KUKA KRL program: MyProgram_128().src

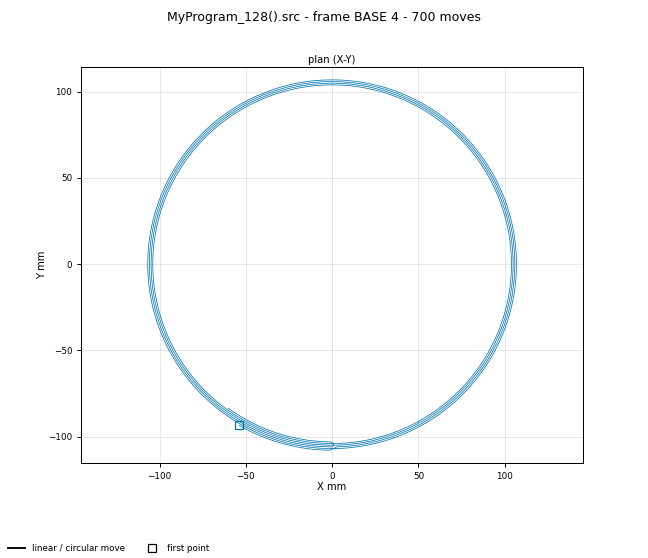
[picture p0: tool path of MyProgram_128().src in frame BASE 4, 700 of 700 moves have a stored position in this frame; points joined in program order, loops and branches not executed]
&ACCESS RVP
&REL 1
&PARAM TEMPLATE = C:\KRC\Roboter\Template\vorgabe
&PARAM EDITMASK = *
DEF MyProgram_128()
; ---- Setting reference (Base) ----
$BASE = BASE_DATA[4]

; --------------------------
; ---- Setting tool (TCP) ----
$TOOL = TOOL_DATA[3]
; --------------------------

$VEL.CP = VEL_APROX_PRINT
Startdeposition()
$VEL.CP = VEL_PRINT
LIN {X -53.8766,Y -93.3824,Z 106,A -123.5845,B 24.9478,C -1.6698,E1 24.9211,E2 209.3121} C_DIS
LIN {X -51.7834,Y -94.56,Z 106,A -122.4157,B 24.9481,C -1.6638,E1 24.9239,E2 208.1542} C_DIS
LIN {X -49.6515,Y -95.6979,Z 106,A -121.0163,B 24.9479,C -1.6666,E1 24.9274,E2 206.7442} C_DIS
LIN {X -46.8609,Y -97.0928,Z 106,A -119.3542,B 24.9481,C -1.6648,E1 24.9316,E2 205.082} C_DIS
LIN {X -43.6897,Y -98.5625,Z 106,A -117.4919,B 24.9481,C -1.6628,E1 24.9363,E2 203.2197} C_DIS
LIN {X -41.2577,Y -99.605,Z 106,A -116.0826,B 24.9483,C -1.6615,E1 24.9399,E2 201.8104} C_DIS
LIN {X -38.8009,Y -100.5875,Z 106,A -114.6732,B 24.9483,C -1.6603,E1 24.9436,E2 200.4009} C_DIS
LIN {X -35.8736,Y -101.6663,Z 106,A -113.2424,B 24.949,C -1.6498,E1 24.9473,E2 198.9921} C_DIS
LIN {X -33.5947,Y -102.4426,Z 106,A -111.8444,B 24.9488,C -1.6534,E1 24.951,E2 197.5829} C_DIS
LIN {X -30.8419,Y -103.3041,Z 106,A -110.1194,B 24.9484,C -1.66,E1 24.9557,E2 195.8392} C_DIS
LIN {X -27.4775,Y -104.2514,Z 106,A -108.3349,B 24.9486,C -1.6559,E1 24.9605,E2 194.0618} C_DIS
LIN {X -24.4492,Y -105.0009,Z 106,A -106.9046,B 24.9492,C -1.6459,E1 24.9643,E2 192.6533} C_DIS
LIN {X -22.329,Y -105.474,Z 106,A -105.5194,B 24.9487,C -1.6546,E1 24.9681,E2 191.2456} C_DIS
LIN {X -19.6263,Y -106.0096,Z 106,A -103.9265,B 24.9484,C -1.6593,E1 24.9725,E2 189.64} C_DIS
LIN {X -15.8193,Y -106.6448,Z 106,A -101.832,B 24.9484,C -1.6604,E1 24.9783,E2 187.5408} C_DIS
LIN {X -12.7268,Y -107.056,Z 106,A -100.4364,B 24.949,C -1.6495,E1 24.9821,E2 186.1701} C_DIS
LIN {X -10.0957,Y -107.3361,Z 106,A -98.9361,B 24.9488,C -1.6532,E1 24.9863,E2 184.6602} C_DIS
LIN {X -7.3812,Y -107.5567,Z 106,A -97.4197,B 24.9486,C -1.656,E1 24.9906,E2 183.1365} C_DIS
LIN {X -3.9682,Y -107.7386,Z 106,A -95.5034,B 24.9483,C -1.6602,E1 24.9959,E2 181.2098} C_DIS
LIN {X -1.323,Y -107.8036,Z 106,A -94.0977,B 24.9483,C -1.6605,E1 24.9999,E2 179.8035} C_DIS
LIN {X -1.323,Y -107.8036,Z 106,A -94.0977,B 24.9483,C -1.6605,E1 24.9999,E2 179.8035} C_DIS
Enddeposition()
LIN {X 0.7537,Y -106.8293,Z 106,A -94.1088,B 24.9501,C -1.6325,E1 24.9997,E2 179.8808} C_DIS
Startdeposition()
$VEL.CP = VEL_PRINT
LIN {X -4.5597,Y -106.7397,Z 106,A -96.7886,B 24.9497,C -1.6389,E1 24.9922,E2 182.546} C_DIS
LIN {X -8.4258,Y -106.5043,Z 106,A -99.1178,B 24.9503,C -1.6288,E1 24.9856,E2 184.8999} C_DIS
LIN {X -12.2598,Y -106.1314,Z 106,A -100.9493,B 24.9497,C -1.6383,E1 24.9806,E2 186.7099} C_DIS
LIN {X -16.8585,Y -105.4999,Z 106,A -103.5719,B 24.95,C -1.6337,E1 24.9733,E2 189.3458} C_DIS
LIN {X -22.5826,Y -104.4233,Z 106,A -106.933,B 24.9505,C -1.6257,E1 24.9641,E2 192.7297} C_DIS
LIN {X -25.8619,Y -103.6611,Z 106,A -108.2155,B 24.9492,C -1.6471,E1 24.9607,E2 193.963} C_DIS
LIN {X -30.0016,Y -102.5389,Z 106,A -110.7389,B 24.9496,C -1.6399,E1 24.9539,E2 196.5076} C_DIS
LIN {X -33.8683,Y -101.3271,Z 106,A -112.9026,B 24.9495,C -1.6419,E1 24.9481,E2 198.6703} C_DIS
LIN {X -37.7546,Y -99.9437,Z 106,A -115.0418,B 24.9492,C -1.6467,E1 24.9425,E2 200.8024} C_DIS
LIN {X -40.9294,Y -98.6879,Z 106,A -117.0692,B 24.9495,C -1.641,E1 24.9373,E2 202.8481} C_DIS
LIN {X -44.6783,Y -97.0474,Z 106,A -120.2088,B 24.9516,C -1.6074,E1 24.9291,E2 206.0752} C_DIS
LIN {X -50.3226,Y -94.2452,Z 106,A -122.6141,B 24.9491,C -1.6488,E1 24.9234,E2 208.3889} C_DIS
LIN {X -53.8043,Y -92.3021,Z 106,A -124.7623,B 24.9489,C -1.6514,E1 24.9181,E2 210.5371} C_DIS
LIN {X -58.2187,Y -89.583,Z 106,A -128.8926,B 24.9517,C -1.6051,E1 24.9082,E2 214.7909} C_DIS
LIN {X -64.5258,Y -85.1515,Z 106,A -131.6457,B 24.9481,C -1.6638,E1 24.9023,E2 217.414} C_DIS
LIN {X -67.7619,Y -82.6008,Z 106,A -133.8259,B 24.9478,C -1.669,E1 24.8975,E2 219.59} C_DIS
LIN {X -70.8575,Y -79.9604,Z 106,A -135.8732,B 24.9472,C -1.6784,E1 24.8932,E2 221.6232} C_DIS
LIN {X -76.0657,Y -75.0211,Z 106,A -139.5928,B 24.9464,C -1.6912,E1 24.8858,E2 225.3276} C_DIS
LIN {X -77.8033,Y -73.2176,Z 106,A -141.1346,B 24.9467,C -1.6867,E1 24.8828,E2 226.8868} C_DIS
LIN {X -80.0433,Y -70.7645,Z 106,A -143.1927,B 24.9471,C -1.6803,E1 24.8789,E2 228.9691} C_DIS
LIN {X -83.2382,Y -66.9754,Z 106,A -146.096,B 24.9473,C -1.6776,E1 24.8737,E2 231.8925} C_DIS
LIN {X -85.3774,Y -64.2251,Z 106,A -147.9105,B 24.9468,C -1.6841,E1 24.8707,E2 233.7001} C_DIS
LIN {X -87.3667,Y -61.4948,Z 106,A -149.2362,B 24.9454,C -1.7066,E1 24.8686,E2 234.9787} C_DIS
LIN {X -89.6712,Y -58.0812,Z 106,A -151.5516,B 24.9454,C -1.7083,E1 24.865,E2 237.3017} C_DIS
LIN {X -91.6677,Y -54.8776,Z 106,A -153.598,B 24.945,C -1.7128,E1 24.862,E2 239.3477} C_DIS
LIN {X -94.7989,Y -49.2714,Z 106,A -156.9611,B 24.9442,C -1.7252,E1 24.8575,E2 242.6992} C_DIS
LIN {X -96.091,Y -46.7001,Z 106,A -158.6935,B 24.9444,C -1.7226,E1 24.8553,E2 244.4471} C_DIS
LIN {X -97.5751,Y -43.5135,Z 106,A -160.5489,B 24.944,C -1.729,E1 24.8532,E2 246.2973} C_DIS
LIN {X -98.9301,Y -40.336,Z 106,A -162.3903,B 24.9436,C -1.7348,E1 24.8512,E2 248.1351} C_DIS
LIN {X -100.5391,Y -36.142,Z 106,A -165.3865,B 24.9445,C -1.7206,E1 24.8483,E2 251.1821} C_DIS
LIN {X -101.8368,Y -32.3055,Z 106,A -167.2873,B 24.9435,C -1.7369,E1 24.8467,E2 253.0548} C_DIS
LIN {X -103.1179,Y -27.944,Z 106,A -169.4189,B 24.9422,C -1.7555,E1 24.8451,E2 255.1546} C_DIS
LIN {X -104.0092,Y -24.4209,Z 106,A -171.4733,B 24.9421,C -1.7577,E1 24.8437,E2 257.2158} C_DIS
LIN {X -104.724,Y -21.1464,Z 106,A -173.1742,B 24.9415,C -1.7668,E1 24.8428,E2 258.905} C_DIS
LIN {X -105.3666,Y -17.6648,Z 106,A -175.1279,B 24.9412,C -1.7708,E1 24.8418,E2 260.8607} C_DIS
LIN {X -105.8765,Y -14.3058,Z 106,A -177.0343,B 24.9411,C -1.7734,E1 24.841,E2 262.7722} C_DIS
LIN {X -106.2835,Y -10.8648,Z 106,A -178.9414,B 24.9408,C -1.7776,E1 24.8405,E2 264.6807} C_DIS
LIN {X -106.6254,Y -6.7385,Z 106,A 178.8379,B 24.9403,C -1.7847,E1 24.84,E2 266.8979} C_DIS
LIN {X -106.7958,Y -2.9825,Z 106,A 176.9449,B 24.9396,C -1.7957,E1 24.8398,E2 268.7761} C_DIS
LIN {X -106.8353,Y 0.6396,Z 106,A 174.8831,B 24.9394,C -1.7977,E1 24.8398,E2 270.8456} C_DIS
LIN {X -106.6524,Y 6.292,Z 106,A 171.4111,B 24.9398,C -1.7917,E1 24.8402,E2 274.3527} C_DIS
LIN {X -106.3816,Y 9.8551,Z 106,A 169.9779,B 24.9382,C -1.8153,E1 24.8406,E2 275.7384} C_DIS
LIN {X -105.9749,Y 13.5463,Z 106,A 167.9438,B 24.9379,C -1.8202,E1 24.8412,E2 277.7729} C_DIS
LIN {X -105.4663,Y 17.0686,Z 106,A 166.0467,B 24.9375,C -1.8267,E1 24.842,E2 279.6657} C_DIS
LIN {X -104.944,Y 20.0236,Z 106,A 164.3886,B 24.9372,C -1.8301,E1 24.8429,E2 281.3254} C_DIS
LIN {X -104.2041,Y 23.5773,Z 106,A 162.302,B 24.9372,C -1.8313,E1 24.8441,E2 283.4215} C_DIS
LIN {X -103.0755,Y 28.1008,Z 106,A 159.897,B 24.9364,C -1.8427,E1 24.8458,E2 285.8133} C_DIS
LIN {X -102.0096,Y 31.7525,Z 106,A 157.8654,B 24.9359,C -1.8494,E1 24.8474,E2 287.8406} C_DIS
LIN {X -100.516,Y 36.206,Z 106,A 155.5457,B 24.9348,C -1.8645,E1 24.8495,E2 290.1376} C_DIS
LIN {X -98.512,Y 41.3469,Z 106,A 152.3947,B 24.9347,C -1.8666,E1 24.8528,E2 293.3012} C_DIS
LIN {X -96.9626,Y 44.8605,Z 106,A 150.3288,B 24.9343,C -1.8726,E1 24.8551,E2 295.3641} C_DIS
LIN {X -95.5,Y 47.8973,Z 106,A 148.3707,B 24.9343,C -1.8726,E1 24.8575,E2 297.3328} C_DIS
LIN {X -93.8185,Y 51.1105,Z 106,A 146.4825,B 24.9337,C -1.8804,E1 24.86,E2 299.2125} C_DIS
LIN {X -91.9159,Y 54.4576,Z 106,A 144.476,B 24.9331,C -1.8885,E1 24.8628,E2 301.2101} C_DIS
LIN {X -90.0123,Y 57.5499,Z 106,A 142.2059,B 24.9336,C -1.8823,E1 24.8662,E2 303.5066} C_DIS
LIN {X -87.3965,Y 61.452,Z 106,A 139.8627,B 24.9326,C -1.8956,E1 24.8699,E2 305.8295} C_DIS
LIN {X -85.1324,Y 64.5512,Z 106,A 137.8079,B 24.9322,C -1.9014,E1 24.8733,E2 307.8805} C_DIS
LIN {X -82.8401,Y 67.4666,Z 106,A 135.7681,B 24.932,C -1.9048,E1 24.8769,E2 309.9218} C_DIS
LIN {X -80.3579,Y 70.4044,Z 106,A 133.8363,B 24.9313,C -1.9149,E1 24.8804,E2 311.8382} C_DIS
LIN {X -78.0201,Y 72.987,Z 106,A 131.9111,B 24.9311,C -1.9175,E1 24.884,E2 313.7657} C_DIS
LIN {X -75.723,Y 75.3681,Z 106,A 130.2361,B 24.9305,C -1.9255,E1 24.8873,E2 315.4289} C_DIS
LIN {X -73.4692,Y 77.5666,Z 106,A 127.978,B 24.9317,C -1.9086,E1 24.8919,E2 317.7366} C_DIS
LIN {X -70.8207,Y 79.9933,Z 106,A 126.0109,B 24.9315,C -1.9115,E1 24.896,E2 319.7045} C_DIS
LIN {X -68.1002,Y 82.32,Z 106,A 124.5718,B 24.9299,C -1.9335,E1 24.899,E2 321.0968} C_DIS
LIN {X -65.2452,Y 84.6004,Z 106,A 122.6715,B 24.9294,C -1.9399,E1 24.9032,E2 322.9889} C_DIS
LIN {X -62.4948,Y 86.6536,Z 106,A 120.7082,B 24.9295,C -1.9391,E1 24.9076,E2 324.9609} C_DIS
LIN {X -59.6356,Y 88.6445,Z 106,A 118.8631,B 24.9292,C -1.9437,E1 24.9118,E2 326.8013} C_DIS
LIN {X -56.8119,Y 90.48,Z 106,A 116.8638,B 24.9294,C -1.94,E1 24.9166,E2 328.8159} C_DIS
LIN {X -53.1715,Y 92.6658,Z 106,A 114.7,B 24.9288,C -1.9483,E1 24.9218,E2 330.9664} C_DIS
LIN {X -49.8424,Y 94.4981,Z 106,A 112.6693,B 24.9286,C -1.952,E1 24.9267,E2 332.9939} C_DIS
LIN {X -46.6974,Y 96.0923,Z 106,A 110.7823,B 24.9283,C -1.9552,E1 24.9315,E2 334.8783} C_DIS
LIN {X -43.2414,Y 97.6968,Z 106,A 108.4552,B 24.9289,C -1.9476,E1 24.9375,E2 337.2292} C_DIS
LIN {X -33.9206,Y 101.3094,Z 106,A 103.3392,B 24.9277,C -1.964,E1 24.9508,E2 342.3169} C_DIS
LIN {X -29.4331,Y 102.7032,Z 106,A 101.1189,B 24.9266,C -1.9783,E1 24.9566,E2 344.507} C_DIS
LIN {X -26.7938,Y 103.4229,Z 106,A 99.4155,B 24.9272,C -1.9707,E1 24.9613,E2 346.2309} C_DIS
LIN {X -23.5828,Y 104.2028,Z 106,A 97.6173,B 24.9272,C -1.9713,E1 24.9661,E2 348.03} C_DIS
LIN {X -19.9636,Y 104.9556,Z 106,A 95.5584,B 24.9272,C -1.9701,E1 24.9718,E2 350.0943} C_DIS
LIN {X -16.1538,Y 105.6089,Z 106,A 93.6037,B 24.9268,C -1.9761,E1 24.9771,E2 352.0365} C_DIS
LIN {X -12.5623,Y 106.096,Z 106,A 91.3704,B 24.9275,C -1.9661,E1 24.9834,E2 354.2952} C_DIS
LIN {X -8.9146,Y 106.4652,Z 106,A 89.0106,B 24.9286,C -1.9518,E1 24.9901,E2 356.6899} C_DIS
LIN {X -4.6596,Y 106.7354,Z 106,A 87.3422,B 24.9268,C -1.9765,E1 24.9946,E2 358.3001} C_DIS
LIN {X 1.7314,Y 106.8233,Z 106,A 84.2326,B 24.9258,C -1.9897,E1 25.0032,E2 361.3784} C_DIS
LIN {X 7.0338,Y 106.6054,Z 106,A 81.2333,B 24.9262,C -1.9838,E1 25.0116,E2 364.3908} C_DIS
LIN {X 12.9512,Y 106.0505,Z 106,A 77.8395,B 24.9268,C -1.9752,E1 25.021,E2 367.8028} C_DIS
LIN {X 16.5164,Y 105.5529,Z 106,A 76.0583,B 24.9264,C -1.9806,E1 25.0259,E2 369.5696} C_DIS
LIN {X 19.8073,Y 104.9856,Z 106,A 74.0743,B 24.9271,C -1.9723,E1 25.0314,E2 371.5712} C_DIS
LIN {X 23.4551,Y 104.2324,Z 106,A 72.1119,B 24.9271,C -1.9727,E1 25.0368,E2 373.5301} C_DIS
LIN {X 26.9434,Y 103.3844,Z 106,A 70.3953,B 24.9265,C -1.9799,E1 25.0414,E2 375.2271} C_DIS
LIN {X 29.9078,Y 102.5667,Z 106,A 68.5867,B 24.9271,C -1.9723,E1 25.0463,E2 377.0505} C_DIS
LIN {X 32.835,Y 101.6662,Z 106,A 66.99,B 24.9271,C -1.9729,E1 25.0505,E2 378.6429} C_DIS
LIN {X 36.1477,Y 100.5373,Z 106,A 65.0474,B 24.9273,C -1.9686,E1 25.0556,E2 380.5918} C_DIS
LIN {X 40.186,Y 98.9912,Z 106,A 62.8015,B 24.9273,C -1.9693,E1 25.0615,E2 382.8313} C_DIS
LIN {X 43.4213,Y 97.6167,Z 106,A 60.1224,B 24.9298,C -1.9351,E1 25.0685,E2 385.5845} C_DIS
LIN {X 47.8384,Y 95.5292,Z 106,A 58.3036,B 24.9277,C -1.9642,E1 25.0729,E2 387.3296} C_DIS
LIN {X 51.0886,Y 93.8304,Z 106,A 56.4015,B 24.9277,C -1.9642,E1 25.0775,E2 389.2263} C_DIS
LIN {X 54.3432,Y 91.9835,Z 106,A 54.3526,B 24.928,C -1.9596,E1 25.0825,E2 391.28} C_DIS
LIN {X 57.4769,Y 90.0591,Z 106,A 52.336,B 24.9284,C -1.9548,E1 25.0873,E2 393.3016} C_DIS
LIN {X 62.2481,Y 86.8297,Z 106,A 49.389,B 24.9284,C -1.9555,E1 25.0941,E2 396.2369} C_DIS
LIN {X 64.5989,Y 85.0966,Z 106,A 47.6628,B 24.929,C -1.9461,E1 25.0979,E2 397.9792} C_DIS
LIN {X 67.8696,Y 82.5116,Z 106,A 45.6524,B 24.9286,C -1.9512,E1 25.1023,E2 399.9698} C_DIS
LIN {X 70.9515,Y 79.8763,Z 106,A 42.9049,B 24.9307,C -1.9232,E1 25.1082,E2 402.7726} C_DIS
LIN {X 73.4992,Y 77.5384,Z 106,A 41.3863,B 24.9299,C -1.9333,E1 25.1112,E2 404.2612} C_DIS
LIN {X 76.148,Y 74.9379,Z 106,A 39.5513,B 24.9298,C -1.9355,E1 25.1148,E2 406.0832} C_DIS
LIN {X 78.2863,Y 72.7037,Z 106,A 37.6743,B 24.9307,C -1.9227,E1 25.1184,E2 407.9824} C_DIS
LIN {X 80.3504,Y 70.4131,Z 106,A 36.1982,B 24.9304,C -1.9264,E1 25.1211,E2 409.4431} C_DIS
LIN {X 82.8244,Y 67.486,Z 106,A 34.1598,B 24.9307,C -1.9222,E1 25.1248,E2 411.4819} C_DIS
LIN {X 85.7964,Y 63.6674,Z 106,A 31.4837,B 24.9314,C -1.9124,E1 25.1293,E2 414.1685} C_DIS
LIN {X 87.8795,Y 60.7571,Z 106,A 29.5343,B 24.9319,C -1.9064,E1 25.1325,E2 416.1227} C_DIS
LIN {X 90.0453,Y 57.4983,Z 106,A 27.5532,B 24.9319,C -1.9059,E1 25.1355,E2 418.0951} C_DIS
LIN {X 92.026,Y 54.2714,Z 106,A 25.5182,B 24.9323,C -1.9003,E1 25.1384,E2 420.1329} C_DIS
LIN {X 94.0721,Y 50.643,Z 106,A 23.5646,B 24.9319,C -1.9061,E1 25.141,E2 422.0625} C_DIS
LIN {X 95.2203,Y 48.4488,Z 106,A 22.0632,B 24.9327,C -1.895,E1 25.143,E2 423.5821} C_DIS
LIN {X 97.1918,Y 44.3641,Z 106,A 19.5636,B 24.9334,C -1.8852,E1 25.146,E2 426.0913} C_DIS
LIN {X 98.6094,Y 41.1158,Z 106,A 17.6218,B 24.9339,C -1.878,E1 25.1481,E2 428.0396} C_DIS
LIN {X 99.9884,Y 37.6368,Z 106,A 15.752,B 24.9339,C -1.878,E1 25.15,E2 429.899} C_DIS
LIN {X 101.4135,Y 33.612,Z 106,A 13.5582,B 24.9341,C -1.8752,E1 25.152,E2 432.087} C_DIS
LIN {X 102.1611,Y 31.2636,Z 106,A 12.0916,B 24.9348,C -1.865,E1 25.1532,E2 433.5693} C_DIS
LIN {X 103.2772,Y 27.3543,Z 106,A 9.9199,B 24.9352,C -1.8587,E1 25.1548,E2 435.7434} C_DIS
LIN {X 104.0784,Y 24.1215,Z 106,A 8.2305,B 24.9353,C -1.8573,E1 25.1559,E2 437.4263} C_DIS
LIN {X 105.1974,Y 18.6478,Z 106,A 4.6721,B 24.9376,C -1.8239,E1 25.1578,E2 441.0428} C_DIS
LIN {X 105.8163,Y 14.7358,Z 106,A 3.0981,B 24.9365,C -1.8406,E1 25.1584,E2 442.568} C_DIS
LIN {X 106.5699,Y 7.559,Z 106,A -0.4908,B 24.9365,C -1.8404,E1 25.1594,E2 446.1362} C_DIS
LIN {X 106.8043,Y 2.7054,Z 106,A -3.4097,B 24.938,C -1.8184,E1 25.1598,E2 449.0895} C_DIS
LIN {X 106.8315,Y -1.2402,Z 106,A -5.5067,B 24.9384,C -1.8124,E1 25.1598,E2 451.1882} C_DIS
LIN {X 106.6676,Y -6.0163,Z 106,A -7.9143,B 24.9385,C -1.8108,E1 25.1595,E2 453.5852} C_DIS
LIN {X 106.4516,Y -9.0849,Z 106,A -9.5091,B 24.9387,C -1.8078,E1 25.1591,E2 455.1777} C_DIS
LIN {X 106.1293,Y -12.2782,Z 106,A -11.3422,B 24.9394,C -1.7974,E1 25.1586,E2 457.0244} C_DIS
LIN {X 105.7046,Y -15.5226,Z 106,A -13.5883,B 24.9412,C -1.7706,E1 25.1577,E2 459.3205} C_DIS
LIN {X 105.0731,Y -19.3387,Z 106,A -15.0265,B 24.9399,C -1.7913,E1 25.157,E2 460.7016} C_DIS
LIN {X 104.3989,Y -22.6941,Z 106,A -16.7856,B 24.94,C -1.7887,E1 25.156,E2 462.4565} C_DIS
LIN {X 103.7322,Y -25.5705,Z 106,A -18.5059,B 24.9408,C -1.7777,E1 25.1549,E2 464.1928} C_DIS
LIN {X 102.7017,Y -29.4385,Z 106,A -20.6789,B 24.9413,C -1.7697,E1 25.1533,E2 466.372} C_DIS
LIN {X 101.627,Y -32.9564,Z 106,A -22.5633,B 24.9415,C -1.7673,E1 25.1517,E2 468.2514} C_DIS
LIN {X 100.5595,Y -36.0867,Z 106,A -24.5742,B 24.9425,C -1.7515,E1 25.1498,E2 470.2883} C_DIS
LIN {X 99.0085,Y -40.1435,Z 106,A -26.6745,B 24.9423,C -1.7542,E1 25.1477,E2 472.3706} C_DIS
LIN {X 97.6883,Y -43.2611,Z 106,A -28.5915,B 24.943,C -1.7443,E1 25.1455,E2 474.3007} C_DIS
LIN {X 96.2281,Y -46.4149,Z 106,A -30.2958,B 24.9429,C -1.7455,E1 25.1435,E2 475.9928} C_DIS
LIN {X 94.0353,Y -50.7107,Z 106,A -32.6182,B 24.9427,C -1.7492,E1 25.1406,E2 478.2943} C_DIS
LIN {X 92.1177,Y -54.1162,Z 106,A -34.9779,B 24.9438,C -1.7317,E1 25.1373,E2 480.6829} C_DIS
LIN {X 90.4395,Y -56.8767,Z 106,A -36.8266,B 24.9444,C -1.7217,E1 25.1345,E2 482.5458} C_DIS
LIN {X 88.6769,Y -59.5878,Z 106,A -38.905,B 24.9457,C -1.7022,E1 25.1312,E2 484.66} C_DIS
LIN {X 86.6097,Y -62.5539,Z 106,A -40.6551,B 24.9455,C -1.7049,E1 25.1284,E2 486.3953} C_DIS
LIN {X 82.7376,Y -67.5931,Z 106,A -43.4459,B 24.9444,C -1.722,E1 25.1237,E2 489.1324} C_DIS
LIN {X 80.2002,Y -70.5851,Z 106,A -45.8759,B 24.9457,C -1.7026,E1 25.1192,E2 491.5971} C_DIS
LIN {X 77.2662,Y -73.7857,Z 106,A -48.251,B 24.9462,C -1.6948,E1 25.1147,E2 493.9805} C_DIS
LIN {X 74.4202,Y -76.6547,Z 106,A -50.3443,B 24.9463,C -1.6926,E1 25.1105,E2 496.07} C_DIS
LIN {X 72.1763,Y -78.7702,Z 106,A -51.968,B 24.9465,C -1.69,E1 25.1072,E2 497.6933} C_DIS
LIN {X 68.8977,Y -81.6549,Z 106,A -54.4497,B 24.9472,C -1.6787,E1 25.1019,E2 500.1919} C_DIS
LIN {X 66.5517,Y -83.5774,Z 106,A -55.9949,B 24.9472,C -1.6786,E1 25.0986,E2 501.7316} C_DIS
LIN {X 63.3055,Y -86.0618,Z 106,A -58.0854,B 24.9472,C -1.6782,E1 25.0939,E2 503.8155} C_DIS
LIN {X 60.6983,Y -87.9203,Z 106,A -59.7674,B 24.9474,C -1.6761,E1 25.0901,E2 505.4965} C_DIS
LIN {X 57.7574,Y -89.879,Z 106,A -61.6475,B 24.9475,C -1.673,E1 25.0857,E2 507.3777} C_DIS
LIN {X 54.914,Y -91.6462,Z 106,A -64.1912,B 24.9497,C -1.6385,E1 25.0795,E2 509.9952} C_DIS
LIN {X 50.9702,Y -93.8946,Z 106,A -66.408,B 24.9494,C -1.6433,E1 25.074,E2 512.1944} C_DIS
LIN {X 47.6133,Y -95.6408,Z 106,A -67.919,B 24.9483,C -1.6614,E1 25.0704,E2 513.6584} C_DIS
LIN {X 44.3076,Y -97.2173,Z 106,A -70.1624,B 24.9492,C -1.6467,E1 25.0646,E2 515.9308} C_DIS
LIN {X 40.356,Y -98.922,Z 106,A -72.1829,B 24.9487,C -1.6552,E1 25.0595,E2 517.9264} C_DIS
LIN {X 37.5686,Y -100.0142,Z 106,A -73.7769,B 24.9487,C -1.6535,E1 25.0553,E2 519.521} C_DIS
LIN {X 34.1433,Y -101.2343,Z 106,A -75.7366,B 24.9489,C -1.6506,E1 25.0502,E2 521.4836} C_DIS
LIN {X 30.0441,Y -102.5263,Z 106,A -78.1285,B 24.9493,C -1.6443,E1 25.0438,E2 523.8861} C_DIS
LIN {X 26.6065,Y -103.471,Z 106,A -79.8614,B 24.949,C -1.6496,E1 25.0391,E2 525.6037} C_DIS
LIN {X 23.3403,Y -104.258,Z 106,A -81.7873,B 24.9494,C -1.6428,E1 25.0338,E2 527.5431} C_DIS
LIN {X 19.8432,Y -104.9787,Z 106,A -83.5686,B 24.9492,C -1.6466,E1 25.029,E2 529.3131} C_DIS
LIN {X 16.582,Y -105.5427,Z 106,A -85.418,B 24.9495,C -1.6423,E1 25.0239,E2 531.1711} C_DIS
LIN {X 9.956,Y -106.3722,Z 106,A -88.9723,B 24.9495,C -1.6412,E1 25.014,E2 534.7253} C_DIS
LIN {X 6.5384,Y -106.6387,Z 106,A -90.9146,B 24.9498,C -1.6361,E1 25.0086,E2 536.6788} C_DIS
LIN {X 3.1284,Y -106.7913,Z 106,A -92.6593,B 24.9497,C -1.6389,E1 25.0037,E2 538.4163} C_DIS
LIN {X 0.7537,Y -106.8293,Z 106,A -94.1068,B 24.9501,C -1.6317,E1 24.9996,E2 539.8808} C_DIS
Enddeposition()
LIN {X 0.7537,Y -106.8293,Z 106,A -94.1068,B 24.9501,C -1.6317,E1 24.9996,E2 539.8808} C_DIS
Startdeposition()
$VEL.CP = VEL_PRINT
LIN {X 2.8627,Y -105.8262,Z 106,A -91.6482,B 24.9457,C -1.7021,E1 25.007,E2 537.2558} C_DIS
LIN {X 7.5893,Y -105.5927,Z 106,A -88.9811,B 24.9454,C -1.7075,E1 25.0144,E2 534.5769} C_DIS
LIN {X 11.0545,Y -105.2857,Z 106,A -87.0189,B 24.9451,C -1.7119,E1 25.0199,E2 532.6057} C_DIS
LIN {X 14.8709,Y -104.8148,Z 106,A -85.4891,B 24.9464,C -1.6906,E1 25.024,E2 531.1276} C_DIS
LIN {X 18.5021,Y -104.2354,Z 106,A -83.6615,B 24.9468,C -1.6855,E1 25.029,E2 529.314} C_DIS
LIN {X 21.3698,Y -103.6852,Z 106,A -81.9293,B 24.9463,C -1.6931,E1 25.0338,E2 527.5658} C_DIS
LIN {X 24.8077,Y -102.9172,Z 106,A -79.9837,B 24.9461,C -1.6965,E1 25.0391,E2 525.6149} C_DIS
LIN {X 27.3407,Y -102.2734,Z 106,A -78.3985,B 24.9455,C -1.705,E1 25.0434,E2 524.0119} C_DIS
LIN {X 30.4857,Y -101.3808,Z 106,A -76.1326,B 24.9441,C -1.7278,E1 25.0496,E2 521.6962} C_DIS
LIN {X 34.7685,Y -99.9926,Z 106,A -74.3733,B 24.9457,C -1.7026,E1 25.0541,E2 520.0001} C_DIS
LIN {X 38.1494,Y -98.7536,Z 106,A -72.4052,B 24.9455,C -1.706,E1 25.0592,E2 518.0281} C_DIS
LIN {X 44.0312,Y -96.275,Z 106,A -68.9082,B 24.945,C -1.7129,E1 25.0682,E2 514.5232} C_DIS
LIN {X 47.5143,Y -94.6044,Z 106,A -66.8339,B 24.9448,C -1.7156,E1 25.0734,E2 512.4479} C_DIS
LIN {X 51.4327,Y -92.5309,Z 106,A -64.1863,B 24.9439,C -1.7303,E1 25.08,E2 509.7733} C_DIS
LIN {X 55.8458,Y -89.9367,Z 106,A -61.8888,B 24.9448,C -1.7155,E1 25.0854,E2 507.5178} C_DIS
LIN {X 60.2465,Y -87.05,Z 106,A -58.7702,B 24.9437,C -1.7326,E1 25.0927,E2 504.3694} C_DIS
LIN {X 63.7862,Y -84.4906,Z 106,A -56.5837,B 24.9439,C -1.73,E1 25.0976,E2 502.1967} C_DIS
LIN {X 68.7462,Y -80.5062,Z 106,A -52.6241,B 24.942,C -1.7597,E1 25.1062,E2 498.182} C_DIS
LIN {X 71.6435,Y -77.9391,Z 106,A -51.0977,B 24.9432,C -1.7403,E1 25.1093,E2 496.7077} C_DIS
LIN {X 74.2627,Y -75.4478,Z 106,A -48.5685,B 24.9413,C -1.7696,E1 25.1144,E2 494.1199} C_DIS
LIN {X 77.038,Y -72.6116,Z 106,A -46.0438,B 24.9399,C -1.7913,E1 25.1193,E2 491.5549} C_DIS
LIN {X 80.7478,Y -68.4627,Z 106,A -44.2008,B 24.9427,C -1.7487,E1 25.1225,E2 489.8208} C_DIS
LIN {X 82.1355,Y -66.7913,Z 106,A -42.1505,B 24.94,C -1.7895,E1 25.1262,E2 487.6839} C_DIS
LIN {X 84.889,Y -63.256,Z 106,A -39.7262,B 24.9395,C -1.7961,E1 25.1303,E2 485.2556} C_DIS
LIN {X 87.4926,Y -59.6021,Z 106,A -37.9624,B 24.941,C -1.7741,E1 25.133,E2 483.5525} C_DIS
LIN {X 89.322,Y -56.8248,Z 106,A -36.1595,B 24.9407,C -1.7793,E1 25.1357,E2 481.7462} C_DIS
LIN {X 91.0435,Y -54.0221,Z 106,A -34.4722,B 24.9406,C -1.7804,E1 25.1381,E2 480.0649} C_DIS
LIN {X 92.6831,Y -51.1605,Z 106,A -32.7776,B 24.9405,C -1.7818,E1 25.1405,E2 478.3759} C_DIS
LIN {X 94.5912,Y -47.5388,Z 106,A -30.0392,B 24.9385,C -1.811,E1 25.144,E2 475.5831} C_DIS
LIN {X 96.0747,Y -44.4634,Z 106,A -28.5555,B 24.9392,C -1.8008,E1 25.1457,E2 474.1315} C_DIS
LIN {X 97.5767,Y -41.0618,Z 106,A -26.9162,B 24.9399,C -1.7908,E1 25.1475,E2 472.5246} C_DIS
LIN {X 99.6096,Y -35.8528,Z 106,A -23.7315,B 24.9388,C -1.807,E1 25.1507,E2 469.3196} C_DIS
LIN {X 100.8837,Y -32.0942,Z 106,A -21.46,B 24.938,C -1.8191,E1 25.1527,E2 467.0324} C_DIS
LIN {X 101.8801,Y -28.7704,Z 106,A -19.6516,B 24.9378,C -1.822,E1 25.1541,E2 465.2273} C_DIS
LIN {X 102.7803,Y -25.3689,Z 106,A -17.7736,B 24.9374,C -1.827,E1 25.1554,E2 463.3486} C_DIS
LIN {X 103.6133,Y -21.7202,Z 106,A -15.6771,B 24.9368,C -1.8365,E1 25.1567,E2 461.2417} C_DIS
LIN {X 104.2406,Y -18.4733,Z 106,A -13.8178,B 24.9362,C -1.8453,E1 25.1576,E2 459.3726} C_DIS
LIN {X 105.3312,Y -10.6197,Z 106,A -9.8154,B 24.9361,C -1.8466,E1 25.1591,E2 455.3908} C_DIS
LIN {X 105.6591,Y -6.5896,Z 106,A -7.3311,B 24.9347,C -1.8665,E1 25.1596,E2 452.8742} C_DIS
LIN {X 105.8662,Y 0.0102,Z 106,A -3.8958,B 24.9343,C -1.872,E1 25.1598,E2 449.4463} C_DIS
LIN {X 105.644,Y 6.8357,Z 106,A -0.212,B 24.9335,C -1.8834,E1 25.1594,E2 445.7576} C_DIS
LIN {X 105.087,Y 12.8161,Z 106,A 2.8902,B 24.9332,C -1.8873,E1 25.1585,E2 442.6645} C_DIS
LIN {X 104.5521,Y 16.6161,Z 106,A 5.3704,B 24.9315,C -1.9114,E1 25.1574,E2 440.1421} C_DIS
LIN {X 103.9962,Y 19.8019,Z 106,A 6.9151,B 24.9318,C -1.908,E1 25.1566,E2 438.6146} C_DIS
LIN {X 103.1739,Y 23.716,Z 106,A 8.8039,B 24.9321,C -1.9028,E1 25.1555,E2 436.749} C_DIS
LIN {X 102.4672,Y 26.605,Z 106,A 10.461,B 24.9316,C -1.9098,E1 25.1544,E2 435.0849} C_DIS
LIN {X 101.6006,Y 29.7448,Z 106,A 12.2454,B 24.9312,C -1.9161,E1 25.153,E2 433.2959} C_DIS
LIN {X 100.3042,Y 33.8577,Z 106,A 15.2868,B 24.9284,C -1.9537,E1 25.1503,E2 430.1829} C_DIS
LIN {X 98.7015,Y 38.282,Z 106,A 17.0851,B 24.9302,C -1.9289,E1 25.1485,E2 428.4532} C_DIS
LIN {X 97.2418,Y 41.8517,Z 106,A 19.906,B 24.9275,C -1.9665,E1 25.1454,E2 425.5589} C_DIS
LIN {X 95.2945,Y 46.1122,Z 106,A 21.697,B 24.9293,C -1.9417,E1 25.1433,E2 423.8362} C_DIS
LIN {X 93.6299,Y 49.4037,Z 106,A 23.5482,B 24.9293,C -1.941,E1 25.1409,E2 421.9963} C_DIS
LIN {X 90.7469,Y 54.5214,Z 106,A 26.8875,B 24.9282,C -1.9564,E1 25.1363,E2 418.6381} C_DIS
LIN {X 89.3815,Y 56.7321,Z 106,A 28.9071,B 24.926,C -1.9863,E1 25.1332,E2 416.5582} C_DIS
LIN {X 86.9485,Y 60.3924,Z 106,A 30.5251,B 24.928,C -1.9599,E1 25.1307,E2 415.0103} C_DIS
LIN {X 85.0327,Y 63.0646,Z 106,A 32.2659,B 24.9278,C -1.9626,E1 25.1278,E2 413.2715} C_DIS
LIN {X 80.7391,Y 68.4729,Z 106,A 36.0206,B 24.9271,C -1.9723,E1 25.1213,E2 409.5115} C_DIS
LIN {X 76.6625,Y 73.0106,Z 106,A 39.4611,B 24.9261,C -1.9855,E1 25.1148,E2 406.055} C_DIS
LIN {X 74.1198,Y 75.589,Z 106,A 41.2078,B 24.9264,C -1.9807,E1 25.1113,E2 404.3269} C_DIS
LIN {X 68.3817,Y 80.8168,Z 106,A 46.1497,B 24.9235,C -2.0201,E1 25.1009,E2 399.3115} C_DIS
LIN {X 65.0054,Y 83.5573,Z 106,A 47.8796,B 24.9251,C -1.9983,E1 25.0972,E2 397.6396} C_DIS
LIN {X 62.5464,Y 85.4121,Z 106,A 49.4512,B 24.9251,C -1.9973,E1 25.0937,E2 396.076} C_DIS
LIN {X 56.181,Y 89.7273,Z 106,A 53.6275,B 24.9247,C -2.0046,E1 25.084,E2 391.8963} C_DIS
LIN {X 51.603,Y 92.436,Z 106,A 56.5544,B 24.9242,C -2.0107,E1 25.0769,E2 388.9638} C_DIS
LIN {X 48.0272,Y 94.3435,Z 106,A 58.6332,B 24.9243,C -2.0089,E1 25.0718,E2 386.8951} C_DIS
LIN {X 42.0104,Y 97.1726,Z 106,A 62.3973,B 24.9235,C -2.0198,E1 25.0622,E2 383.1147} C_DIS
LIN {X 38.4539,Y 98.6339,Z 106,A 64.5154,B 24.9232,C -2.0235,E1 25.0567,E2 380.9928} C_DIS
LIN {X 34.2369,Y 100.1764,Z 106,A 66.8535,B 24.9233,C -2.0219,E1 25.0506,E2 378.6632} C_DIS
LIN {X 30.9143,Y 101.2512,Z 106,A 68.7609,B 24.9232,C -2.0241,E1 25.0455,E2 376.7542} C_DIS
LIN {X 27.6976,Y 102.177,Z 106,A 70.7839,B 24.9224,C -2.0338,E1 25.04,E2 374.7113} C_DIS
LIN {X 23.2873,Y 103.2729,Z 106,A 72.9882,B 24.9231,C -2.0249,E1 25.034,E2 372.5313} C_DIS
LIN {X 19.9726,Y 103.9634,Z 106,A 74.751,B 24.9233,C -2.0229,E1 25.0292,E2 370.7753} C_DIS
LIN {X 16.3742,Y 104.5907,Z 106,A 76.7722,B 24.9231,C -2.0253,E1 25.0237,E2 368.7504} C_DIS
LIN {X 12.6191,Y 105.1101,Z 106,A 78.5481,B 24.9239,C -2.0149,E1 25.0188,E2 367.0008} C_DIS
LIN {X 9.519,Y 105.4358,Z 106,A 80.5849,B 24.9228,C -2.0289,E1 25.0131,E2 364.932} C_DIS
LIN {X 2.137,Y 105.8431,Z 106,A 84.243,B 24.9239,C -2.0152,E1 25.003,E2 361.3077} C_DIS
LIN {X -3.1739,Y 105.8169,Z 106,A 87.1486,B 24.9239,C -2.0157,E1 24.9949,E2 358.4008} C_DIS
LIN {X -8.4104,Y 105.5299,Z 106,A 90.209,B 24.9232,C -2.0232,E1 24.9863,E2 355.3216} C_DIS
LIN {X -11.8336,Y 105.2017,Z 106,A 92.1844,B 24.923,C -2.0266,E1 24.9807,E2 353.3369} C_DIS
LIN {X -15.8704,Y 104.6686,Z 106,A 94.2832,B 24.9234,C -2.0211,E1 24.975,E2 351.2494} C_DIS
LIN {X -19.0255,Y 104.1412,Z 106,A 95.9121,B 24.9238,C -2.0159,E1 24.9705,E2 349.6314} C_DIS
LIN {X -23.6859,Y 103.1808,Z 106,A 98.554,B 24.9238,C -2.0162,E1 24.9633,E2 346.9855} C_DIS
LIN {X -27.059,Y 102.3495,Z 106,A 100.5723,B 24.9235,C -2.0196,E1 24.9578,E2 344.9561} C_DIS
LIN {X -33.227,Y 100.5168,Z 106,A 103.871,B 24.9244,C -2.0086,E1 24.9491,E2 341.6779} C_DIS
LIN {X -36.8621,Y 99.2399,Z 106,A 106.4985,B 24.923,C -2.0267,E1 24.942,E2 339.0022} C_DIS
LIN {X -40.0141,Y 98.0111,Z 106,A 107.8505,B 24.9246,C -2.0059,E1 24.9387,E2 337.6968} C_DIS
LIN {X -42.6877,Y 96.8773,Z 106,A 109.4161,B 24.9247,C -2.0033,E1 24.9346,E2 336.1335} C_DIS
LIN {X -45.5288,Y 95.5748,Z 106,A 111.258,B 24.9245,C -2.0064,E1 24.93,E2 334.2796} C_DIS
LIN {X -48.9379,Y 93.8753,Z 106,A 113.2934,B 24.9248,C -2.002,E1 24.9249,E2 332.2491} C_DIS
LIN {X -52.0537,Y 92.1843,Z 106,A 115.144,B 24.9253,C -1.9961,E1 24.9204,E2 330.4073} C_DIS
LIN {X -56.7908,Y 89.3438,Z 106,A 118.1999,B 24.9255,C -1.9931,E1 24.9131,E2 327.3492} C_DIS
LIN {X -59.0447,Y 87.87,Z 106,A 119.6867,B 24.9256,C -1.9913,E1 24.9097,E2 325.8616} C_DIS
LIN {X -62.0878,Y 85.7479,Z 106,A 121.755,B 24.9258,C -1.9895,E1 24.905,E2 323.7906} C_DIS
LIN {X -64.9051,Y 83.6346,Z 106,A 123.6632,B 24.9261,C -1.9855,E1 24.9007,E2 321.8848} C_DIS
LIN {X -68.1739,Y 80.9939,Z 106,A 125.9502,B 24.9264,C -1.981,E1 24.8958,E2 319.6} C_DIS
LIN {X -70.9992,Y 78.5268,Z 106,A 128.3426,B 24.9258,C -1.9898,E1 24.8908,E2 317.1769} C_DIS
LIN {X -73.5191,Y 76.1724,Z 106,A 129.7662,B 24.9273,C -1.9689,E1 24.888,E2 315.7972} C_DIS
LIN {X -76.0564,Y 73.6394,Z 106,A 131.7184,B 24.9276,C -1.9646,E1 24.8842,E2 313.8469} C_DIS
LIN {X -78.5004,Y 71.0301,Z 106,A 133.7226,B 24.9278,C -1.9623,E1 24.8804,E2 311.8394} C_DIS
LIN {X -80.8451,Y 68.3485,Z 106,A 135.6945,B 24.9281,C -1.959,E1 24.8768,E2 309.8665} C_DIS
LIN {X -83.1469,Y 65.5279,Z 106,A 137.6052,B 24.9286,C -1.9516,E1 24.8735,E2 307.9645} C_DIS
LIN {X -85.4044,Y 62.557,Z 106,A 139.6282,B 24.929,C -1.9462,E1 24.8701,E2 305.9445} C_DIS
LIN {X -87.6141,Y 59.4228,Z 106,A 142.3682,B 24.9276,C -1.965,E1 24.8657,E2 303.1463} C_DIS
LIN {X -89.9799,Y 55.7766,Z 106,A 144.1356,B 24.9297,C -1.9367,E1 24.8631,E2 301.4373} C_DIS
LIN {X -91.9047,Y 52.5438,Z 106,A 146.1991,B 24.93,C -1.9318,E1 24.8602,E2 299.3747} C_DIS
LIN {X -93.7537,Y 49.1687,Z 106,A 148.2951,B 24.9304,C -1.9262,E1 24.8575,E2 297.2811} C_DIS
LIN {X -94.954,Y 46.809,Z 106,A 150.2712,B 24.9293,C -1.9418,E1 24.855,E2 295.2569} C_DIS
LIN {X -96.7172,Y 43.0501,Z 106,A 152.0193,B 24.9311,C -1.9167,E1 24.8531,E2 293.5592} C_DIS
LIN {X -97.7488,Y 40.6535,Z 106,A 153.7003,B 24.9307,C -1.9222,E1 24.8512,E2 291.8557} C_DIS
LIN {X -99.5097,Y 36.1265,Z 106,A 156.4958,B 24.9309,C -1.9201,E1 24.8485,E2 289.0494} C_DIS
LIN {X -100.7038,Y 32.6501,Z 106,A 158.1312,B 24.9323,C -1.901,E1 24.8471,E2 287.4503} C_DIS
LIN {X -101.8094,Y 29.0201,Z 106,A 160.5744,B 24.9317,C -1.9087,E1 24.8452,E2 284.9745} C_DIS
LIN {X -102.7697,Y 25.4123,Z 106,A 162.2001,B 24.9332,C -1.8878,E1 24.8441,E2 283.3891} C_DIS
LIN {X -103.5908,Y 21.8295,Z 106,A 164.105,B 24.9339,C -1.8784,E1 24.843,E2 281.4955} C_DIS
LIN {X -104.2053,Y 18.6691,Z 106,A 165.8484,B 24.9342,C -1.8729,E1 24.8421,E2 279.755} C_DIS
LIN {X -104.7782,Y 15.1282,Z 106,A 167.7677,B 24.9347,C -1.8658,E1 24.8413,E2 277.8412} C_DIS
LIN {X -105.1798,Y 12.0242,Z 106,A 169.6239,B 24.9347,C -1.8662,E1 24.8406,E2 275.9728} C_DIS
LIN {X -105.4706,Y 9.1428,Z 106,A 171.1767,B 24.9351,C -1.8606,E1 24.8403,E2 274.4241} C_DIS
LIN {X -105.7264,Y 5.4137,Z 106,A 173.5452,B 24.9347,C -1.8667,E1 24.8399,E2 272.0269} C_DIS
LIN {X -105.8434,Y 2.1194,Z 106,A 174.9213,B 24.9361,C -1.846,E1 24.8399,E2 270.6917} C_DIS
LIN {X -105.8565,Y -1.4057,Z 106,A 176.9162,B 24.9363,C -1.843,E1 24.8399,E2 268.6921} C_DIS
LIN {X -105.7439,Y -5.0782,Z 106,A 178.9586,B 24.9366,C -1.8386,E1 24.8401,E2 266.6479} C_DIS
LIN {X -105.5037,Y -8.7372,Z 106,A -179.0558,B 24.9371,C -1.8323,E1 24.8405,E2 264.6654} C_DIS
LIN {X -105.1493,Y -12.2844,Z 106,A -177.195,B 24.9377,C -1.8236,E1 24.841,E2 262.814} C_DIS
LIN {X -104.6518,Y -15.9788,Z 106,A -175.1557,B 24.938,C -1.818,E1 24.8418,E2 260.7759} C_DIS
LIN {X -104.0557,Y -19.4929,Z 106,A -173.0977,B 24.9381,C -1.8167,E1 24.8429,E2 258.709} C_DIS
LIN {X -103.481,Y -22.3388,Z 106,A -171.0979,B 24.9374,C -1.8275,E1 24.8441,E2 256.6716} C_DIS
LIN {X -102.5941,Y -26.1113,Z 106,A -169.5132,B 24.9391,C -1.8022,E1 24.8451,E2 255.138} C_DIS
LIN {X -101.8265,Y -28.9597,Z 106,A -167.4342,B 24.9382,C -1.8151,E1 24.8467,E2 253.0163} C_DIS
LIN {X -100.7666,Y -32.4559,Z 106,A -166.107,B 24.9403,C -1.7852,E1 24.8478,E2 251.7526} C_DIS
LIN {X -98.9819,Y -37.5483,Z 106,A -162.9931,B 24.9403,C -1.7836,E1 24.8507,E2 248.625} C_DIS
LIN {X -97.685,Y -40.8049,Z 106,A -161.0817,B 24.9407,C -1.7786,E1 24.8527,E2 246.7149} C_DIS
LIN {X -96.3823,Y -43.7932,Z 106,A -159.2198,B 24.9408,C -1.7771,E1 24.8549,E2 244.8461} C_DIS
LIN {X -94.5322,Y -47.6581,Z 106,A -157.033,B 24.9416,C -1.7657,E1 24.8575,E2 242.6748} C_DIS
LIN {X -92.2919,Y -51.861,Z 106,A -154.2953,B 24.9416,C -1.7646,E1 24.8612,E2 239.9253} C_DIS
LIN {X -90.3984,Y -55.0947,Z 106,A -152.2969,B 24.9421,C -1.7581,E1 24.8641,E2 237.932} C_DIS
LIN {X -88.507,Y -58.0848,Z 106,A -150.4341,B 24.9425,C -1.7512,E1 24.8669,E2 236.0762} C_DIS
LIN {X -86.5882,Y -60.9107,Z 106,A -148.052,B 24.9415,C -1.7665,E1 24.8708,E2 233.6461} C_DIS
LIN {X -84.447,Y -63.8437,Z 106,A -146.3282,B 24.9424,C -1.7526,E1 24.8736,E2 231.947} C_DIS
LIN {X -81.5652,Y -67.4867,Z 106,A -144.3313,B 24.9441,C -1.7273,E1 24.877,E2 230.0011} C_DIS
LIN {X -78.7064,Y -70.8,Z 106,A -141.5738,B 24.9435,C -1.7364,E1 24.8822,E2 227.2094} C_DIS
LIN {X -75.8967,Y -73.8051,Z 106,A -139.0996,B 24.9432,C -1.7409,E1 24.887,E2 224.7138} C_DIS
LIN {X -71.0216,Y -78.5081,Z 106,A -135.6885,B 24.9443,C -1.7237,E1 24.8939,E2 221.3298} C_DIS
LIN {X -68.6891,Y -80.5549,Z 106,A -134.0153,B 24.9445,C -1.7202,E1 24.8974,E2 219.6583} C_DIS
LIN {X -65.722,Y -82.9935,Z 106,A -131.9806,B 24.9449,C -1.7147,E1 24.9018,E2 217.6291} C_DIS
LIN {X -63.7704,Y -84.5025,Z 106,A -130.0605,B 24.9436,C -1.7348,E1 24.9062,E2 215.6544} C_DIS
LIN {X -60.5255,Y -86.856,Z 106,A -128.2986,B 24.9449,C -1.7154,E1 24.9101,E2 213.9325} C_DIS
LIN {X -56.6041,Y -89.4627,Z 106,A -125.6929,B 24.9449,C -1.7136,E1 24.9163,E2 211.3227} C_DIS
LIN {X -53.0814,Y -91.5958,Z 106,A -123.5078,B 24.9453,C -1.7087,E1 24.9215,E2 209.1426} C_DIS
LIN {X -49.4012,Y -93.6313,Z 106,A -120.7152,B 24.9442,C -1.7258,E1 24.9285,E2 206.3015} C_DIS
LIN {X -45.4356,Y -95.6196,Z 106,A -118.7593,B 24.9455,C -1.7055,E1 24.9333,E2 204.3888} C_DIS
LIN {X -41.6456,Y -97.3307,Z 106,A -116.8523,B 24.9465,C -1.6897,E1 24.9381,E2 202.5149} C_DIS
LIN {X -39.357,Y -98.2782,Z 106,A -115.3197,B 24.9461,C -1.6958,E1 24.9421,E2 200.9643} C_DIS
LIN {X -36.2456,Y -99.4663,Z 106,A -113.5485,B 24.9463,C -1.693,E1 24.9467,E2 199.1962} C_DIS
LIN {X -32.7817,Y -100.6612,Z 106,A -111.5778,B 24.9464,C -1.6909,E1 24.952,E2 197.2268} C_DIS
LIN {X -30.4278,Y -101.398,Z 106,A -110.0375,B 24.946,C -1.698,E1 24.9561,E2 195.667} C_DIS
LIN {X -26.4858,Y -102.4978,Z 106,A -108.072,B 24.9467,C -1.6868,E1 24.9614,E2 193.7251} C_DIS
LIN {X -23.0076,Y -103.3351,Z 106,A -106.0102,B 24.9464,C -1.6908,E1 24.967,E2 191.6512} C_DIS
LIN {X -17.9021,Y -104.3408,Z 106,A -103.1967,B 24.9465,C -1.6896,E1 24.9747,E2 188.8374} C_DIS
LIN {X -15.3096,Y -104.7525,Z 106,A -101.1784,B 24.945,C -1.7133,E1 24.9805,E2 186.7613} C_DIS
LIN {X -10.9746,Y -105.2941,Z 106,A -99.3436,B 24.9464,C -1.6916,E1 24.9854,E2 184.9767} C_DIS
LIN {X -6.0849,Y -105.6897,Z 106,A -96.9191,B 24.947,C -1.6824,E1 24.9921,E2 182.5733} C_DIS
LIN {X -0.0735,Y -105.866,Z 106,A -93.7201,B 24.947,C -1.6806,E1 25.0011,E2 179.3782} C_DIS
LIN {X -0.0735,Y -105.866,Z 106,A -93.7201,B 24.947,C -1.6806,E1 25.0011,E2 179.3782} C_DIS
Enddeposition()
LIN {X 0.7394,Y -104.8869,Z 106,A -94.0052,B 24.9478,C -1.6689,E1 25.0002,E2 179.6911} C_DIS
Startdeposition()
$VEL.CP = VEL_PRINT
LIN {X -4.1892,Y -104.8087,Z 106,A -96.5208,B 24.9474,C -1.6754,E1 24.9932,E2 182.1915} C_DIS
LIN {X -10.0388,Y -104.4111,Z 106,A -99.7415,B 24.9474,C -1.6746,E1 24.9842,E2 185.4152} C_DIS
LIN {X -14.0541,Y -103.9475,Z 106,A -102.1585,B 24.9479,C -1.6668,E1 24.9775,E2 187.8524} C_DIS
LIN {X -17.4636,Y -103.428,Z 106,A -103.8774,B 24.9475,C -1.6738,E1 24.9728,E2 189.5563} C_DIS
LIN {X -23.5123,Y -102.2227,Z 106,A -107.3728,B 24.9477,C -1.6703,E1 24.9632,E2 193.0641} C_DIS
LIN {X -27.1829,Y -101.3086,Z 106,A -109.1052,B 24.9468,C -1.6843,E1 24.9586,E2 194.7657} C_DIS
LIN {X -31.5521,Y -100.0351,Z 106,A -112.0031,B 24.9477,C -1.6702,E1 24.9507,E2 197.7019} C_DIS
LIN {X -34.713,Y -98.9814,Z 106,A -113.6437,B 24.9472,C -1.6786,E1 24.9464,E2 199.3258} C_DIS
LIN {X -37.7682,Y -97.8584,Z 106,A -115.7309,B 24.9478,C -1.6685,E1 24.9409,E2 201.4414} C_DIS
LIN {X -41.7226,Y -96.2371,Z 106,A -117.811,B 24.9471,C -1.6806,E1 24.9356,E2 203.4975} C_DIS
LIN {X -44.1583,Y -95.1439,Z 106,A -120.1357,B 24.949,C -1.6498,E1 24.9295,E2 205.9013} C_DIS
LIN {X -48.5561,Y -92.9771,Z 106,A -122.0555,B 24.947,C -1.6814,E1 24.9249,E2 207.751} C_DIS
LIN {X -52.8383,Y -90.6135,Z 106,A -124.5883,B 24.9465,C -1.6903,E1 24.9188,E2 210.2699} C_DIS
LIN {X -54.9785,Y -89.3303,Z 106,A -126.0876,B 24.9467,C -1.6873,E1 24.9152,E2 211.7812} C_DIS
LIN {X -57.6685,Y -87.6165,Z 106,A -127.8319,B 24.9465,C -1.6899,E1 24.9111,E2 213.5249} C_DIS
LIN {X -63.0852,Y -83.8008,Z 106,A -131.4468,B 24.9461,C -1.6962,E1 24.9029,E2 217.1373} C_DIS
LIN {X -66.0157,Y -81.5122,Z 106,A -133.5394,B 24.946,C -1.6977,E1 24.8983,E2 219.2342} C_DIS
LIN {X -68.9702,Y -79.028,Z 106,A -135.602,B 24.9456,C -1.7034,E1 24.8939,E2 221.2911} C_DIS
LIN {X -70.8987,Y -77.3025,Z 106,A -138.2636,B 24.9483,C -1.661,E1 24.8883,E2 224.0647} C_DIS
LIN {X -75.6281,Y -72.6823,Z 106,A -140.154,B 24.9438,C -1.7312,E1 24.8849,E2 225.7959} C_DIS
LIN {X -79.641,Y -68.2621,Z 106,A -143.9327,B 24.9446,C -1.7195,E1 24.8777,E2 229.6191} C_DIS
LIN {X -81.7637,Y -65.7053,Z 106,A -145.702,B 24.9442,C -1.7255,E1 24.8746,E2 231.3825} C_DIS
LIN {X -83.0881,Y -64.0208,Z 106,A -147.6463,B 24.9458,C -1.7004,E1 24.8712,E2 233.3958} C_DIS
LIN {X -85.8097,Y -60.3266,Z 106,A -149.5015,B 24.9439,C -1.7301,E1 24.8683,E2 235.1895} C_DIS
LIN {X -87.8791,Y -57.2703,Z 106,A -151.6526,B 24.9439,C -1.7304,E1 24.8649,E2 237.3506} C_DIS
LIN {X -90.1718,Y -53.5855,Z 106,A -153.7076,B 24.9427,C -1.748,E1 24.862,E2 239.374} C_DIS
LIN {X -92.1341,Y -50.1361,Z 106,A -156.1526,B 24.943,C -1.7439,E1 24.8586,E2 241.8416} C_DIS
LIN {X -94.5359,Y -45.4452,Z 106,A -158.8936,B 24.9421,C -1.7569,E1 24.8552,E2 244.5664} C_DIS
LIN {X -96.0234,Y -42.2126,Z 106,A -160.9127,B 24.942,C -1.7597,E1 24.8529,E2 246.5899} C_DIS
LIN {X -97.4211,Y -38.8814,Z 106,A -162.9615,B 24.9418,C -1.7628,E1 24.8507,E2 248.6429} C_DIS
LIN {X -99.3304,Y -33.7019,Z 106,A -166.984,B 24.9435,C -1.7363,E1 24.8469,E2 252.7513} C_DIS
LIN {X -101.0878,Y -27.999,Z 106,A -170.3232,B 24.943,C -1.7435,E1 24.8444,E2 256.0928} C_DIS
LIN {X -102.54,Y -22.0888,Z 106,A -172.3048,B 24.9392,C -1.801,E1 24.8433,E2 257.949} C_DIS
LIN {X -103.1139,Y -19.2404,Z 106,A -174.2566,B 24.9397,C -1.793,E1 24.8422,E2 259.9314} C_DIS
LIN {X -103.7289,Y -15.5829,Z 106,A -176.221,B 24.9392,C -1.8015,E1 24.8414,E2 261.887} C_DIS
LIN {X -104.1598,Y -12.3724,Z 106,A -177.9949,B 24.9388,C -1.807,E1 24.8408,E2 263.6585} C_DIS
LIN {X -104.5336,Y -8.6674,Z 106,A 179.9702,B 24.9384,C -1.8135,E1 24.8402,E2 265.6901} C_DIS
LIN {X -104.7641,Y -5.2084,Z 106,A 177.9398,B 24.9383,C -1.8147,E1 24.8399,E2 267.7298} C_DIS
LIN {X -104.8792,Y -1.6561,Z 106,A 176.1222,B 24.9375,C -1.8253,E1 24.8398,E2 269.533} C_DIS
LIN {X -104.8732,Y 1.9797,Z 106,A 174.2424,B 24.9368,C -1.8355,E1 24.8398,E2 271.3999} C_DIS
LIN {X -104.553,Y 8.4253,Z 106,A 170.6043,B 24.9363,C -1.8429,E1 24.8404,E2 275.0422} C_DIS
LIN {X -104.2547,Y 11.5616,Z 106,A 168.7378,B 24.9363,C -1.8433,E1 24.8409,E2 276.9189} C_DIS
LIN {X -103.799,Y 15.1059,Z 106,A 166.7974,B 24.9358,C -1.85,E1 24.8417,E2 278.8549} C_DIS
LIN {X -103.2715,Y 18.3666,Z 106,A 165.1424,B 24.9351,C -1.8611,E1 24.8424,E2 280.4933} C_DIS
LIN {X -102.687,Y 21.396,Z 106,A 163.4493,B 24.9347,C -1.8662,E1 24.8434,E2 282.1842} C_DIS
LIN {X -101.8642,Y 25.0204,Z 106,A 160.7729,B 24.9358,C -1.85,E1 24.8451,E2 284.9149} C_DIS
LIN {X -100.8836,Y 28.7197,Z 106,A 159.2093,B 24.9341,C -1.8751,E1 24.8463,E2 286.4277} C_DIS
LIN {X -98.5216,Y 35.9974,Z 106,A 155.2164,B 24.9327,C -1.8947,E1 24.8498,E2 290.3967} C_DIS
LIN {X -96.9837,Y 39.9584,Z 106,A 152.7501,B 24.9326,C -1.8967,E1 24.8523,E2 292.8721} C_DIS
LIN {X -95.4225,Y 43.5558,Z 106,A 150.2086,B 24.9331,C -1.8891,E1 24.8552,E2 295.4457} C_DIS
LIN {X -92.4829,Y 49.493,Z 106,A 146.7916,B 24.9318,C -1.907,E1 24.8595,E2 298.8384} C_DIS
LIN {X -90.8087,Y 52.4991,Z 106,A 144.4523,B 24.9326,C -1.8962,E1 24.8628,E2 301.2155} C_DIS
LIN {X -88.8826,Y 55.6975,Z 106,A 142.3553,B 24.9323,C -1.9,E1 24.8659,E2 303.3141} C_DIS
LIN {X -86.7328,Y 58.9896,Z 106,A 140.7156,B 24.9306,C -1.9239,E1 24.8684,E2 304.905} C_DIS
LIN {X -84.796,Y 61.7415,Z 106,A 138.9562,B 24.93,C -1.9318,E1 24.8713,E2 306.6543} C_DIS
LIN {X -82.9443,Y 64.2075,Z 106,A 137.1271,B 24.93,C -1.9311,E1 24.8744,E2 308.4936} C_DIS
LIN {X -80.6568,Y 67.058,Z 106,A 135.211,B 24.9295,C -1.9393,E1 24.8777,E2 310.3992} C_DIS
LIN {X -78.3421,Y 69.7488,Z 106,A 133.2575,B 24.9292,C -1.9437,E1 24.8813,E2 312.351} C_DIS
LIN {X -76.0945,Y 72.1952,Z 106,A 131.3587,B 24.9291,C -1.9452,E1 24.885,E2 314.2545} C_DIS
LIN {X -73.6835,Y 74.6529,Z 106,A 129.5499,B 24.9285,C -1.9523,E1 24.8885,E2 316.0539} C_DIS
LIN {X -68.2484,Y 79.6527,Z 106,A 125.576,B 24.9277,C -1.9638,E1 24.8967,E2 320.0164} C_DIS
LIN {X -65.9951,Y 81.5289,Z 106,A 123.8916,B 24.9277,C -1.9644,E1 24.9003,E2 321.706} C_DIS
LIN {X -63.0696,Y 83.8125,Z 106,A 121.8632,B 24.9273,C -1.9686,E1 24.9048,E2 323.7316} C_DIS
LIN {X -60.1368,Y 85.9417,Z 106,A 119.7157,B 24.9275,C -1.9666,E1 24.9097,E2 325.8914} C_DIS
LIN {X -56.675,Y 88.2624,Z 106,A 116.5262,B 24.9296,C -1.938,E1 24.9174,E2 329.1591} C_DIS
LIN {X -51.6451,Y 91.2985,Z 106,A 114.2328,B 24.9267,C -1.9768,E1 24.9228,E2 331.3671} C_DIS
LIN {X -48.3695,Y 93.0754,Z 106,A 112.2036,B 24.9265,C -1.9805,E1 24.9277,E2 333.3932} C_DIS
LIN {X -44.7869,Y 94.8513,Z 106,A 109.8025,B 24.9268,C -1.976,E1 24.9338,E2 335.8112} C_DIS
LIN {X -40.8134,Y 96.626,Z 106,A 107.7085,B 24.9258,C -1.9899,E1 24.9391,E2 337.8771} C_DIS
LIN {X -34.1174,Y 99.1903,Z 106,A 103.8498,B 24.9252,C -1.9971,E1 24.9492,E2 341.7265} C_DIS
LIN {X -28.1244,Y 101.0523,Z 106,A 100.2833,B 24.9253,C -1.9958,E1 24.9587,E2 345.3022} C_DIS
LIN {X -25.3911,Y 101.7737,Z 106,A 97.933,B 24.9274,C -1.9674,E1 24.9653,E2 347.7233} C_DIS
LIN {X -20.3375,Y 102.9026,Z 106,A 95.9368,B 24.9249,C -2.0007,E1 24.9706,E2 349.6426} C_DIS
LIN {X -17.106,Y 103.4878,Z 106,A 94.1403,B 24.9249,C -2.002,E1 24.9755,E2 351.438} C_DIS
LIN {X -13.8806,Y 103.9702,Z 106,A 92.2591,B 24.925,C -1.9993,E1 24.9807,E2 353.327} C_DIS
LIN {X -9.9051,Y 104.4235,Z 106,A 90.1766,B 24.9247,C -2.0044,E1 24.9865,E2 355.3986} C_DIS
LIN {X -4.877,Y 104.7791,Z 106,A 87.3761,B 24.9247,C -2.0037,E1 24.9943,E2 358.2017} C_DIS
LIN {X -0.503,Y 104.8908,Z 106,A 85.061,B 24.9245,C -2.0072,E1 25.0007,E2 360.5087} C_DIS
LIN {X 2.8751,Y 104.853,Z 106,A 82.6071,B 24.9262,C -1.9842,E1 25.0077,E2 363.0167} C_DIS
LIN {X 6.9566,Y 104.661,Z 106,A 81.247,B 24.9237,C -2.0176,E1 25.0113,E2 364.297} C_DIS
LIN {X 10.8223,Y 104.3321,Z 106,A 78.9022,B 24.9243,C -2.0086,E1 25.0179,E2 366.6617} C_DIS
LIN {X 14.2036,Y 103.9272,Z 106,A 77.0166,B 24.9245,C -2.0072,E1 25.0231,E2 368.5491} C_DIS
LIN {X 17.065,Y 103.4947,Z 106,A 75.4338,B 24.9245,C -2.0067,E1 25.0275,E2 370.1317} C_DIS
LIN {X 20.6307,Y 102.844,Z 106,A 73.441,B 24.9245,C -2.0054,E1 25.0329,E2 372.1254} C_DIS
LIN {X 24.1354,Y 102.0788,Z 106,A 71.6239,B 24.9243,C -2.0099,E1 25.0378,E2 373.9292} C_DIS
LIN {X 28.7234,Y 100.8825,Z 106,A 68.8691,B 24.9249,C -2.0018,E1 25.0453,E2 376.699} C_DIS
LIN {X 32.7258,Y 99.6571,Z 106,A 66.4302,B 24.9255,C -1.994,E1 25.0518,E2 379.1518} C_DIS
LIN {X 37.5299,Y 97.9488,Z 106,A 63.8505,B 24.925,C -1.9995,E1 25.0586,E2 381.713} C_DIS
LIN {X 40.9979,Y 96.5482,Z 106,A 60.9314,B 24.9278,C -1.9628,E1 25.0663,E2 384.712} C_DIS
LIN {X 45.7078,Y 94.4097,Z 106,A 58.8998,B 24.9257,C -1.9907,E1 25.0712,E2 386.6723} C_DIS
LIN {X 49.5977,Y 92.4261,Z 106,A 56.6561,B 24.9255,C -1.9932,E1 25.0768,E2 388.9039} C_DIS
LIN {X 53.4465,Y 90.254,Z 106,A 54.1788,B 24.926,C -1.9872,E1 25.0828,E2 391.3879} C_DIS
LIN {X 55.9575,Y 88.7202,Z 106,A 51.6819,B 24.9288,C -1.9492,E1 25.0889,E2 393.9667} C_DIS
LIN {X 60.4325,Y 85.7356,Z 106,A 49.6226,B 24.9265,C -1.9794,E1 25.0934,E2 395.9475} C_DIS
LIN {X 63.1231,Y 83.7724,Z 106,A 47.9528,B 24.9263,C -1.9823,E1 25.0971,E2 397.6046} C_DIS
LIN {X 66.7085,Y 80.9473,Z 106,A 45.3232,B 24.9271,C -1.9721,E1 25.1029,E2 400.2484} C_DIS
LIN {X 70.1135,Y 78.0157,Z 106,A 42.3012,B 24.9291,C -1.9443,E1 25.1093,E2 403.3241} C_DIS
LIN {X 73.2416,Y 75.089,Z 106,A 40.4924,B 24.9279,C -1.9609,E1 25.1129,E2 405.0863} C_DIS
LIN {X 77.6544,Y 70.5152,Z 106,A 37.0691,B 24.9283,C -1.9552,E1 25.1194,E2 408.5081} C_DIS
LIN {X 79.9004,Y 67.9576,Z 106,A 34.3104,B 24.9313,C -1.9142,E1 25.1246,E2 411.3509} C_DIS
LIN {X 83.4772,Y 63.5159,Z 106,A 32.1277,B 24.9291,C -1.9447,E1 25.1282,E2 413.4515} C_DIS
LIN {X 85.4727,Y 60.8009,Z 106,A 30.4816,B 24.9288,C -1.9481,E1 25.1308,E2 415.0814} C_DIS
LIN {X 88.8774,Y 55.7058,Z 106,A 27.1946,B 24.9293,C -1.942,E1 25.1359,E2 418.3666} C_DIS
LIN {X 91.9516,Y 50.4726,Z 106,A 23.726,B 24.9304,C -1.9266,E1 25.1408,E2 421.8535} C_DIS
LIN {X 93.4921,Y 47.556,Z 106,A 21.9387,B 24.9307,C -1.9222,E1 25.1431,E2 423.6417} C_DIS
LIN {X 94.5841,Y 45.3448,Z 106,A 19.6315,B 24.9338,C -1.8787,E1 25.1459,E2 426.0391} C_DIS
LIN {X 96.9014,Y 40.1597,Z 106,A 17.5669,B 24.9314,C -1.9127,E1 25.1481,E2 428.0123} C_DIS
LIN {X 99.195,Y 34.1034,Z 106,A 13.6016,B 24.9334,C -1.8843,E1 25.1519,E2 432.0223} C_DIS
LIN {X 100.1895,Y 31.0541,Z 106,A 12.2688,B 24.9326,C -1.8966,E1 25.153,E2 433.3186} C_DIS
LIN {X 101.1871,Y 27.6325,Z 106,A 10.4167,B 24.9327,C -1.8946,E1 25.1544,E2 435.1648} C_DIS
LIN {X 101.9958,Y 24.481,Z 106,A 8.4928,B 24.9335,C -1.8829,E1 25.1557,E2 437.1051} C_DIS
LIN {X 102.7662,Y 21.0101,Z 106,A 5.634,B 24.9366,C -1.8386,E1 25.1574,E2 440.0517} C_DIS
LIN {X 103.7701,Y 15.3094,Z 106,A 3.4268,B 24.9346,C -1.8684,E1 25.1583,E2 442.1756} C_DIS
LIN {X 104.2395,Y 11.6916,Z 106,A 0.847,B 24.9367,C -1.8375,E1 25.1591,E2 444.8131} C_DIS
LIN {X 104.6342,Y 7.3537,Z 106,A -0.5627,B 24.9344,C -1.8706,E1 25.1594,E2 446.1363} C_DIS
LIN {X 104.8762,Y 1.8176,Z 106,A -3.7133,B 24.9355,C -1.8556,E1 25.1598,E2 449.3037} C_DIS
LIN {X 104.8883,Y -0.9201,Z 106,A -5.804,B 24.9375,C -1.8257,E1 25.1598,E2 451.4525} C_DIS
LIN {X 104.7964,Y -4.4748,Z 106,A -7.7845,B 24.9381,C -1.8178,E1 25.1595,E2 453.4398} C_DIS
LIN {X 104.5662,Y -8.2592,Z 106,A -9.3397,B 24.937,C -1.8328,E1 25.1592,E2 454.9504} C_DIS
LIN {X 104.2718,Y -11.398,Z 106,A -12.1102,B 24.9404,C -1.7832,E1 25.1583,E2 457.8214} C_DIS
LIN {X 103.4484,Y -17.3416,Z 106,A -14.2272,B 24.9378,C -1.8213,E1 25.1574,E2 459.8362} C_DIS
LIN {X 102.8306,Y -20.6962,Z 106,A -16.0187,B 24.938,C -1.8183,E1 25.1565,E2 461.6243} C_DIS
LIN {X 101.9708,Y -24.5835,Z 106,A -18.3127,B 24.9388,C -1.8063,E1 25.1551,E2 463.9333} C_DIS
LIN {X 101.0418,Y -28.1613,Z 106,A -20.3294,B 24.9393,C -1.8,E1 25.1536,E2 465.9533} C_DIS
LIN {X 100.136,Y -31.2268,Z 106,A -22.6442,B 24.9412,C -1.7705,E1 25.1516,E2 468.3243} C_DIS
LIN {X 98.8071,Y -35.2096,Z 106,A -24.1331,B 24.9395,C -1.7972,E1 25.1503,E2 469.7419} C_DIS
LIN {X 96.604,Y -40.8656,Z 106,A -27.5362,B 24.9404,C -1.7832,E1 25.1468,E2 473.1591} C_DIS
LIN {X 93.8298,Y -46.8851,Z 106,A -31.5406,B 24.9422,C -1.7561,E1 25.142,E2 477.2059} C_DIS
LIN {X 91.6327,Y -51.0468,Z 106,A -33.6993,B 24.9416,C -1.7658,E1 25.1392,E2 479.3305} C_DIS
LIN {X 89.9458,Y -53.9668,Z 106,A -35.4653,B 24.9417,C -1.7637,E1 25.1367,E2 481.0925} C_DIS
LIN {X 88.3614,Y -56.5208,Z 106,A -37.2144,B 24.9423,C -1.7545,E1 25.1341,E2 482.8544} C_DIS
LIN {X 86.4441,Y -59.4141,Z 106,A -39.5334,B 24.9438,C -1.7314,E1 25.1303,E2 485.2163} C_DIS
LIN {X 84.5115,Y -62.1301,Z 106,A -41.7874,B 24.9453,C -1.7086,E1 25.1265,E2 487.5135} C_DIS
LIN {X 81.3269,Y -66.2443,Z 106,A -43.7692,B 24.9435,C -1.7367,E1 25.1232,E2 489.4197} C_DIS
LIN {X 76.8735,Y -71.3658,Z 106,A -47.2629,B 24.9435,C -1.736,E1 25.1168,E2 492.8993} C_DIS
LIN {X 72.7177,Y -75.594,Z 106,A -51.5922,B 24.9469,C -1.683,E1 25.108,E2 497.3354} C_DIS
LIN {X 68.6443,Y -79.3126,Z 106,A -53.3281,B 24.944,C -1.7287,E1 25.1046,E2 498.9567} C_DIS
LIN {X 65.0624,Y -82.2751,Z 106,A -56.1284,B 24.9451,C -1.7122,E1 25.0985,E2 501.7853} C_DIS
LIN {X 59.9,Y -86.1063,Z 106,A -60.0166,B 24.9465,C -1.6893,E1 25.0896,E2 505.7137} C_DIS
LIN {X 55.5602,Y -88.9684,Z 106,A -62.4807,B 24.9459,C -1.6992,E1 25.0839,E2 508.1464} C_DIS
LIN {X 52.2952,Y -90.9259,Z 106,A -65.5443,B 24.9486,C -1.6554,E1 25.0763,E2 511.3042} C_DIS
LIN {X 47.3372,Y -93.6039,Z 106,A -67.6651,B 24.9465,C -1.6889,E1 25.0712,E2 513.3399} C_DIS
LIN {X 44.2032,Y -95.123,Z 106,A -70.0231,B 24.9479,C -1.6675,E1 25.0651,E2 515.7427} C_DIS
LIN {X 40.8566,Y -96.6078,Z 106,A -72.0112,B 24.9481,C -1.665,E1 25.06,E2 517.7319} C_DIS
LIN {X 37.4604,Y -97.9752,Z 106,A -74.8998,B 24.9504,C -1.6269,E1 25.0522,E2 520.7045} C_DIS
LIN {X 30.6189,Y -100.3245,Z 106,A -77.1465,B 24.9465,C -1.6902,E1 25.0467,E2 522.7973} C_DIS
LIN {X 26.6327,Y -101.4559,Z 106,A -79.8164,B 24.9477,C -1.6713,E1 25.0394,E2 525.5075} C_DIS
LIN {X 22.852,Y -102.3736,Z 106,A -81.8517,B 24.9476,C -1.6729,E1 25.0339,E2 527.5363} C_DIS
LIN {X 19.358,Y -103.0912,Z 106,A -83.8381,B 24.9478,C -1.6697,E1 25.0284,E2 529.5279} C_DIS
LIN {X 15.7977,Y -103.6957,Z 106,A -85.6736,B 24.9475,C -1.6737,E1 25.0234,E2 531.352} C_DIS
LIN {X 8.0985,Y -104.5791,Z 106,A -90.0048,B 24.9479,C -1.6673,E1 25.0113,E2 535.6954} C_DIS
LIN {X 5.148,Y -104.7673,Z 106,A -92.2059,B 24.9494,C -1.6436,E1 25.005,E2 537.9518} C_DIS
LIN {X 1.0715,Y -104.8873,Z 106,A -93.9854,B 24.9483,C -1.6605,E1 25.0002,E2 539.6911} C_DIS
LIN {X 1.0715,Y -104.8873,Z 106,A -93.9854,B 24.9483,C -1.6605,E1 25.0002,E2 539.6911} C_DIS
Enddeposition()
LIN {X 0.7371,Y -103.9038,Z 106,A -93.865,B 24.9465,C -1.6897,E1 25.0007,E2 539.5014} C_DIS
Startdeposition()
$VEL.CP = VEL_PRINT
LIN {X 4.6847,Y -103.8139,Z 106,A -91.1086,B 24.945,C -1.7129,E1 25.0086,E2 536.6905} C_DIS
LIN {X 8.0211,Y -103.6096,Z 106,A -89.1325,B 24.9446,C -1.7191,E1 25.0141,E2 534.7008} C_DIS
LIN {X 14.2586,Y -102.9371,Z 106,A -85.7105,B 24.9446,C -1.7196,E1 25.0236,E2 531.28} C_DIS
LIN {X 17.5278,Y -102.4312,Z 106,A -83.9225,B 24.9446,C -1.7196,E1 25.0285,E2 529.494} C_DIS
LIN {X 20.8525,Y -101.8056,Z 106,A -82.067,B 24.9446,C -1.7208,E1 25.0336,E2 527.6378} C_DIS
LIN {X 24.0331,Y -101.1039,Z 106,A -80.1308,B 24.944,C -1.7281,E1 25.0389,E2 525.6869} C_DIS
LIN {X 30.7665,Y -99.2604,Z 106,A -76.0089,B 24.943,C -1.7435,E1 25.05,E2 521.5355} C_DIS
LIN {X 33.8948,Y -98.2368,Z 106,A -74.2027,B 24.943,C -1.7455,E1 25.0548,E2 519.7283} C_DIS
LIN {X 36.9168,Y -97.141,Z 106,A -73.0012,B 24.9443,C -1.7246,E1 25.0578,E2 518.5788} C_DIS
LIN {X 39.4363,Y -96.1461,Z 106,A -70.9668,B 24.9427,C -1.7488,E1 25.0632,E2 516.4917} C_DIS
LIN {X 44.3753,Y -93.9701,Z 106,A -68.4753,B 24.9437,C -1.7335,E1 25.0694,E2 514.0426} C_DIS
LIN {X 47.1075,Y -92.6291,Z 106,A -66.1247,B 24.9417,C -1.764,E1 25.0755,E2 511.6263} C_DIS
LIN {X 50.6084,Y -90.7635,Z 106,A -64.9112,B 24.9441,C -1.7277,E1 25.0782,E2 510.502} C_DIS
LIN {X 53.8398,Y -88.8848,Z 106,A -62.4955,B 24.9429,C -1.7461,E1 25.0841,E2 508.0503} C_DIS
LIN {X 56.4082,Y -87.2779,Z 106,A -60.8814,B 24.9429,C -1.747,E1 25.0879,E2 506.4393} C_DIS
LIN {X 59.5534,Y -85.1627,Z 106,A -58.4013,B 24.9415,C -1.7674,E1 25.0937,E2 503.9195} C_DIS
LIN {X 62.822,Y -82.782,Z 106,A -56.4687,B 24.942,C -1.7597,E1 25.098,E2 502.0119} C_DIS
LIN {X 65.5918,Y -80.6038,Z 106,A -54.5221,B 24.9417,C -1.7642,E1 25.1022,E2 500.0621} C_DIS
LIN {X 68.7411,Y -77.9367,Z 106,A -51.808,B 24.9401,C -1.7878,E1 25.108,E2 497.303} C_DIS
LIN {X 71.4202,Y -75.4882,Z 106,A -50.4178,B 24.9415,C -1.7669,E1 25.1108,E2 495.9677} C_DIS
LIN {X 73.6829,Y -73.2814,Z 106,A -48.3759,B 24.9404,C -1.7837,E1 25.1149,E2 493.8948} C_DIS
LIN {X 76.8681,Y -69.9336,Z 106,A -45.6305,B 24.9394,C -1.7985,E1 25.1201,E2 491.1266} C_DIS
LIN {X 79.0455,Y -67.4613,Z 106,A -44.5596,B 24.9412,C -1.7719,E1 25.1219,E2 490.1233} C_DIS
LIN {X 80.7368,Y -65.4277,Z 106,A -42.7273,B 24.9399,C -1.7914,E1 25.1252,E2 488.2534} C_DIS
LIN {X 84.1329,Y -61.0008,Z 106,A -39.5733,B 24.9391,C -1.803,E1 25.1306,E2 485.0871} C_DIS
LIN {X 85.8824,Y -58.5109,Z 106,A -38.0661,B 24.9392,C -1.8005,E1 25.1329,E2 483.5932} C_DIS
LIN {X 87.6072,Y -55.8952,Z 106,A -36.4165,B 24.9392,C -1.8021,E1 25.1354,E2 481.9481} C_DIS
LIN {X 89.046,Y -53.5746,Z 106,A -34.8428,B 24.9386,C -1.8093,E1 25.1377,E2 480.3654} C_DIS
LIN {X 90.7186,Y -50.6888,Z 106,A -33.0331,B 24.9384,C -1.8135,E1 25.1402,E2 478.5552} C_DIS
LIN {X 94.1329,Y -44.0255,Z 106,A -29.2492,B 24.9385,C -1.8112,E1 25.145,E2 474.7968} C_DIS
LIN {X 95.2622,Y -41.5249,Z 106,A -27.4337,B 24.9373,C -1.8286,E1 25.147,E2 472.9502} C_DIS
LIN {X 97.045,Y -37.1704,Z 106,A -24.7659,B 24.9366,C -1.8397,E1 25.1498,E2 470.2709} C_DIS
LIN {X 99.3428,Y -30.5009,Z 106,A -21.3028,B 24.937,C -1.8338,E1 25.1529,E2 466.8414} C_DIS
LIN {X 100.0066,Y -28.2473,Z 106,A -19.7418,B 24.9359,C -1.8491,E1 25.1541,E2 465.2531} C_DIS
LIN {X 101.06,Y -24.2112,Z 106,A -17.2534,B 24.9348,C -1.8645,E1 25.1558,E2 462.7429} C_DIS
LIN {X 101.9683,Y -20.0459,Z 106,A -15.0416,B 24.9348,C -1.8661,E1 25.1571,E2 460.5401} C_DIS
LIN {X 102.5644,Y -16.7308,Z 106,A -12.6003,B 24.9325,C -1.8971,E1 25.1582,E2 458.0401} C_DIS
LIN {X 103.1583,Y -12.5618,Z 106,A -11.1063,B 24.9345,C -1.8692,E1 25.1587,E2 456.6206} C_DIS
LIN {X 103.5968,Y -8.1813,Z 106,A -8.546,B 24.9335,C -1.8828,E1 25.1594,E2 454.0435} C_DIS
LIN {X 103.8509,Y -3.8229,Z 106,A -5.6284,B 24.9314,C -1.9123,E1 25.1598,E2 451.0736} C_DIS
LIN {X 103.9197,Y -0.2336,Z 106,A -4.2977,B 24.933,C -1.8911,E1 25.1598,E2 449.8009} C_DIS
LIN {X 103.893,Y 2.3826,Z 106,A -2.0577,B 24.9302,C -1.9297,E1 25.1596,E2 447.483} C_DIS
LIN {X 103.7037,Y 6.6979,Z 106,A -0.5572,B 24.9323,C -1.8998,E1 25.1594,E2 446.062} C_DIS
LIN {X 103.3589,Y 10.7772,Z 106,A 1.4819,B 24.9325,C -1.8979,E1 25.1589,E2 444.0397} C_DIS
LIN {X 103.1222,Y 12.8559,Z 106,A 3.1494,B 24.9307,C -1.9232,E1 25.1583,E2 442.3221} C_DIS
LIN {X 102.626,Y 16.3506,Z 106,A 5.5319,B 24.9289,C -1.948,E1 25.1573,E2 439.8953} C_DIS
LIN {X 101.9209,Y 20.2913,Z 106,A 7.1183,B 24.9303,C -1.9285,E1 25.1565,E2 438.3642} C_DIS
LIN {X 101.2357,Y 23.4637,Z 106,A 8.9556,B 24.9297,C -1.9361,E1 25.1553,E2 436.5196} C_DIS
LIN {X 100.3605,Y 26.9632,Z 106,A 10.8847,B 24.9295,C -1.9397,E1 25.154,E2 434.5932} C_DIS
LIN {X 99.4076,Y 30.292,Z 106,A 13.4661,B 24.9269,C -1.974,E1 25.1519,E2 431.9456} C_DIS
LIN {X 98.0777,Y 34.3509,Z 106,A 15.0513,B 24.9288,C -1.9484,E1 25.1505,E2 430.4295} C_DIS
LIN {X 96.6572,Y 38.1658,Z 106,A 17.3037,B 24.9283,C -1.9554,E1 25.1483,E2 428.1733} C_DIS
LIN {X 95.3402,Y 41.346,Z 106,A 19.8286,B 24.926,C -1.9873,E1 25.1454,E2 425.5869} C_DIS
LIN {X 93.7013,Y 44.9364,Z 106,A 21.0391,B 24.9285,C -1.9529,E1 25.1441,E2 424.4641} C_DIS
LIN {X 91.9486,Y 48.4218,Z 106,A 23.5371,B 24.927,C -1.9734,E1 25.1409,E2 421.9311} C_DIS
LIN {X 89.3158,Y 53.1223,Z 106,A 26.2809,B 24.927,C -1.9719,E1 25.1371,E2 419.2049} C_DIS
LIN {X 88.1274,Y 55.0706,Z 106,A 27.7773,B 24.9261,C -1.9852,E1 25.1349,E2 417.6849} C_DIS
LIN {X 85.1504,Y 59.5712,Z 106,A 30.5621,B 24.9261,C -1.9849,E1 25.1306,E2 414.9145} C_DIS
LIN {X 83.6374,Y 61.6777,Z 106,A 32.137,B 24.9254,C -1.9944,E1 25.1279,E2 413.3247} C_DIS
LIN {X 80.0404,Y 66.278,Z 106,A 35.2684,B 24.9251,C -1.9985,E1 25.1225,E2 410.1983} C_DIS
LIN {X 78.0844,Y 68.572,Z 106,A 37.0723,B 24.9244,C -2.0082,E1 25.1192,E2 408.3798} C_DIS
LIN {X 74.0989,Y 72.8603,Z 106,A 40.0443,B 24.9246,C -2.0048,E1 25.1135,E2 405.4288} C_DIS
LIN {X 72.0436,Y 74.8929,Z 106,A 42.7545,B 24.9209,C -2.0542,E1 25.1079,E2 402.613} C_DIS
LIN {X 67.9655,Y 78.6141,Z 106,A 44.5798,B 24.9242,C -2.01,E1 25.1043,E2 400.8993} C_DIS
LIN {X 65.0035,Y 81.0806,Z 106,A 47.1719,B 24.9225,C -2.0331,E1 25.0986,E2 398.2626} C_DIS
LIN {X 61.3324,Y 83.8901,Z 106,A 49.4893,B 24.9229,C -2.0282,E1 25.0934,E2 395.965} C_DIS
LIN {X 56.5217,Y 87.205,Z 106,A 52.7679,B 24.9223,C -2.0358,E1 25.0858,E2 392.6795} C_DIS
LIN {X 53.756,Y 88.9358,Z 106,A 54.5847,B 24.922,C -2.0392,E1 25.0815,E2 390.8602} C_DIS
LIN {X 50.0653,Y 91.0661,Z 106,A 56.9519,B 24.9217,C -2.0432,E1 25.0757,E2 388.4906} C_DIS
LIN {X 47.156,Y 92.6043,Z 106,A 58.4185,B 24.9226,C -2.0317,E1 25.0722,E2 387.0553} C_DIS
LIN {X 44.7391,Y 93.7961,Z 106,A 60.6101,B 24.9203,C -2.0618,E1 25.0665,E2 384.7983} C_DIS
LIN {X 41.4802,Y 95.2818,Z 106,A 61.6455,B 24.923,C -2.0265,E1 25.0641,E2 383.8489} C_DIS
LIN {X 38.1732,Y 96.6543,Z 106,A 64.0946,B 24.9214,C -2.0474,E1 25.0576,E2 381.356} C_DIS
LIN {X 35.1351,Y 97.8008,Z 106,A 65.8831,B 24.9213,C -2.049,E1 25.0529,E2 379.5675} C_DIS
LIN {X 31.0571,Y 99.1703,Z 106,A 67.9447,B 24.9221,C -2.0387,E1 25.0476,E2 377.5342} C_DIS
LIN {X 28.1982,Y 100.0205,Z 106,A 70.4158,B 24.9195,C -2.0725,E1 25.0407,E2 374.9871} C_DIS
LIN {X 24.4417,Y 101.0042,Z 106,A 72.0372,B 24.9209,C -2.0532,E1 25.0365,E2 373.4139} C_DIS
LIN {X 20.863,Y 101.8034,Z 106,A 73.9558,B 24.9212,C -2.0502,E1 25.0312,E2 371.505} C_DIS
LIN {X 17.4751,Y 102.44,Z 106,A 75.9684,B 24.9208,C -2.0552,E1 25.0257,E2 369.4825} C_DIS
LIN {X 13.6291,Y 103.022,Z 106,A 78.068,B 24.9208,C -2.054,E1 25.0199,E2 367.3876} C_DIS
LIN {X 10.0678,Y 103.4317,Z 106,A 80.2096,B 24.9204,C -2.0607,E1 25.0139,E2 365.2315} C_DIS
LIN {X 6.3687,Y 103.7258,Z 106,A 82.4049,B 24.9199,C -2.0666,E1 25.0077,E2 363.0234} C_DIS
LIN {X 1.6776,Y 103.906,Z 106,A 84.583,B 24.9212,C -2.0505,E1 25.0018,E2 360.884} C_DIS
LIN {X -1.0881,Y 103.9146,Z 106,A 86.2205,B 24.9209,C -2.0544,E1 24.9972,E2 359.237} C_DIS
LIN {X -5.6849,Y 103.7637,Z 106,A 88.8371,B 24.9207,C -2.0567,E1 24.9899,E2 356.6144} C_DIS
LIN {X -9.5536,Y 103.4792,Z 106,A 90.8193,B 24.9212,C -2.0498,E1 24.9844,E2 354.6479} C_DIS
LIN {X -12.6755,Y 103.145,Z 106,A 92.838,B 24.9204,C -2.0597,E1 24.9787,E2 352.6043} C_DIS
LIN {X -17.1002,Y 102.5027,Z 106,A 95.035,B 24.9214,C -2.0478,E1 24.9727,E2 350.4335} C_DIS
LIN {X -20.5394,Y 101.8699,Z 106,A 98.2771,B 24.9176,C -2.0964,E1 24.9636,E2 347.0723} C_DIS
LIN {X -27.0282,Y 100.3429,Z 106,A 100.4804,B 24.9222,C -2.0368,E1 24.958,E2 345.0074} C_DIS
LIN {X -34.1951,Y 98.1324,Z 106,A 104.5525,B 24.9228,C -2.0296,E1 24.9472,E2 340.9454} C_DIS
LIN {X -38.3407,Y 96.5885,Z 106,A 107.1878,B 24.9225,C -2.0336,E1 24.9402,E2 338.295} C_DIS
LIN {X -41.0248,Y 95.4803,Z 106,A 109.0443,B 24.9219,C -2.0408,E1 24.9354,E2 336.4171} C_DIS
LIN {X -44.766,Y 93.7832,Z 106,A 111.4326,B 24.9219,C -2.0419,E1 24.9293,E2 334.0202} C_DIS
LIN {X -48.4813,Y 91.9173,Z 106,A 113.4276,B 24.923,C -2.0271,E1 24.9244,E2 332.055} C_DIS
LIN {X -52.5658,Y 89.6436,Z 106,A 116.3979,B 24.9222,C -2.037,E1 24.9172,E2 329.0523} C_DIS
LIN {X -56.7146,Y 87.0805,Z 106,A 118.6262,B 24.9239,C -2.015,E1 24.912,E2 326.8694} C_DIS
LIN {X -59.3171,Y 85.327,Z 106,A 120.5249,B 24.9237,C -2.0177,E1 24.9076,E2 324.9577} C_DIS
LIN {X -62.4122,Y 83.0899,Z 106,A 122.6145,B 24.924,C -2.0128,E1 24.9029,E2 322.8726} C_DIS
LIN {X -65.3994,Y 80.7598,Z 106,A 124.6749,B 24.9245,C -2.0072,E1 24.8984,E2 320.8177} C_DIS
LIN {X -68.1955,Y 78.4132,Z 106,A 127.2379,B 24.9233,C -2.0227,E1 24.8929,E2 318.2077} C_DIS
LIN {X -70.9453,Y 75.9348,Z 106,A 128.7763,B 24.925,C -1.9997,E1 24.8898,E2 316.7181} C_DIS
LIN {X -73.2847,Y 73.6796,Z 106,A 130.5518,B 24.9254,C -1.9948,E1 24.8863,E2 314.9467} C_DIS
LIN {X -75.7401,Y 71.1523,Z 106,A 132.5061,B 24.9257,C -1.9904,E1 24.8825,E2 312.9943} C_DIS
LIN {X -78.0642,Y 68.5951,Z 106,A 134.4612,B 24.9259,C -1.9874,E1 24.8789,E2 311.0378} C_DIS
LIN {X -80.3507,Y 65.9041,Z 106,A 136.5083,B 24.9261,C -1.9859,E1 24.8752,E2 308.9848} C_DIS
LIN {X -82.6066,Y 63.0523,Z 106,A 138.525,B 24.9264,C -1.9809,E1 24.8718,E2 306.9703} C_DIS
LIN {X -84.6911,Y 60.2217,Z 106,A 140.3301,B 24.9272,C -1.9709,E1 24.8688,E2 305.1804} C_DIS
LIN {X -87.1563,Y 56.5976,Z 106,A 143.8736,B 24.9246,C -2.0048,E1 24.8633,E2 301.5383} C_DIS
LIN {X -90.1929,Y 51.6187,Z 106,A 146.1052,B 24.928,C -1.96,E1 24.8603,E2 299.4019} C_DIS
LIN {X -93.4415,Y 45.4773,Z 106,A 149.9876,B 24.9287,C -1.9504,E1 24.8553,E2 295.5216} C_DIS
LIN {X -94.9297,Y 42.2819,Z 106,A 151.7649,B 24.9295,C -1.9386,E1 24.8533,E2 293.7627} C_DIS
LIN {X -96.0074,Y 39.7767,Z 106,A 153.67,B 24.9288,C -1.9483,E1 24.8512,E2 291.8239} C_DIS
LIN {X -97.5433,Y 35.8411,Z 106,A 156.3096,B 24.9285,C -1.9522,E1 24.8486,E2 289.16} C_DIS
LIN {X -98.852,Y 32.0547,Z 106,A 157.6445,B 24.9313,C -1.9142,E1 24.8475,E2 287.9082} C_DIS
LIN {X -99.5803,Y 29.7153,Z 106,A 159.2884,B 24.9309,C -1.9203,E1 24.8461,E2 286.2402} C_DIS
LIN {X -100.5291,Y 26.3315,Z 106,A 161.3026,B 24.9311,C -1.9169,E1 24.8447,E2 284.2225} C_DIS
LIN {X -101.6623,Y 21.5479,Z 106,A 163.8957,B 24.932,C -1.9041,E1 24.8431,E2 281.6449} C_DIS
LIN {X -102.2937,Y 18.3089,Z 106,A 165.78,B 24.9323,C -1.9005,E1 24.8421,E2 279.7578} C_DIS
LIN {X -102.8616,Y 14.79,Z 106,A 167.7914,B 24.9326,C -1.8958,E1 24.8412,E2 277.7456} C_DIS
LIN {X -103.3255,Y 11.0967,Z 106,A 169.8443,B 24.9331,C -1.8892,E1 24.8406,E2 275.6962} C_DIS
LIN {X -103.6347,Y 7.7073,Z 106,A 172.2345,B 24.9322,C -1.9014,E1 24.84,E2 273.2626} C_DIS
LIN {X -103.835,Y 4.1927,Z 106,A 173.4435,B 24.9345,C -1.8692,E1 24.84,E2 272.1233} C_DIS
LIN {X -103.9027,Y 1.8584,Z 106,A 174.9843,B 24.9342,C -1.874,E1 24.8398,E2 270.5617} C_DIS
LIN {X -103.9057,Y -1.6916,Z 106,A 177.0202,B 24.9344,C -1.8704,E1 24.8398,E2 268.522} C_DIS
LIN {X -103.7693,Y -5.5834,Z 106,A 179.118,B 24.935,C -1.8618,E1 24.8401,E2 266.4322} C_DIS
LIN {X -103.5258,Y -9.0489,Z 106,A -178.8772,B 24.9352,C -1.8588,E1 24.8405,E2 264.4224} C_DIS
LIN {X -103.169,Y -12.471,Z 106,A -177.0182,B 24.9357,C -1.8514,E1 24.8411,E2 262.5699} C_DIS
LIN {X -102.7018,Y -15.8604,Z 106,A -175.1277,B 24.9361,C -1.8456,E1 24.8419,E2 260.682} C_DIS
LIN {X -102.0819,Y -19.4563,Z 106,A -173.0091,B 24.9363,C -1.8431,E1 24.8429,E2 258.5568} C_DIS
LIN {X -100.8032,Y -25.2594,Z 106,A -169.7758,B 24.9371,C -1.8314,E1 24.845,E2 255.3324} C_DIS
LIN {X -100.0323,Y -28.1565,Z 106,A -168.122,B 24.9375,C -1.8264,E1 24.8462,E2 253.681} C_DIS
LIN {X -98.23,Y -33.9168,Z 106,A -164.656,B 24.9378,C -1.8213,E1 24.8492,E2 250.2072} C_DIS
LIN {X -97.227,Y -36.6897,Z 106,A -163.1702,B 24.9385,C -1.8115,E1 24.8506,E2 248.7365} C_DIS
LIN {X -96.0251,Y -39.7332,Z 106,A -161.2581,B 24.9385,C -1.8101,E1 24.8526,E2 246.817} C_DIS
LIN {X -94.6774,Y -42.8419,Z 106,A -159.4212,B 24.939,C -1.8037,E1 24.8547,E2 244.9854} C_DIS
LIN {X -92.343,Y -47.6673,Z 106,A -156.7448,B 24.9403,C -1.7853,E1 24.858,E2 242.3383} C_DIS
LIN {X -90.0465,Y -51.8735,Z 106,A -154.1585,B 24.9409,C -1.7761,E1 24.8615,E2 239.7604} C_DIS
LIN {X -88.888,Y -53.8346,Z 106,A -152.5882,B 24.9403,C -1.7841,E1 24.8637,E2 238.1629} C_DIS
LIN {X -87.0407,Y -56.775,Z 106,A -150.5611,B 24.9404,C -1.7832,E1 24.8668,E2 236.1277} C_DIS
LIN {X -85.0313,Y -59.7425,Z 106,A -148.2713,B 24.94,C -1.7897,E1 24.8705,E2 233.8113} C_DIS
LIN {X -82.7027,Y -62.9276,Z 106,A -146.4621,B 24.9412,C -1.7709,E1 24.8735,E2 232.0381} C_DIS
LIN {X -80.5887,Y -65.6105,Z 106,A -144.6284,B 24.9416,C -1.7646,E1 24.8766,E2 230.2106} C_DIS
LIN {X -78.2934,Y -68.3327,Z 106,A -142.0358,B 24.9404,C -1.7833,E1 24.8815,E2 227.5618} C_DIS
LIN {X -75.6789,Y -71.2174,Z 106,A -140.6723,B 24.9426,C -1.7497,E1 24.8839,E2 226.2724} C_DIS
LIN {X -73.8446,Y -73.1178,Z 106,A -138.3051,B 24.9406,C -1.7802,E1 24.8888,E2 223.8223} C_DIS
LIN {X -70.6828,Y -76.1806,Z 106,A -136.4577,B 24.9424,C -1.7537,E1 24.8924,E2 222.0307} C_DIS
LIN {X -67.8943,Y -78.6763,Z 106,A -134.3633,B 24.9426,C -1.7508,E1 24.8968,E2 219.9349} C_DIS
LIN {X -65.0245,Y -81.0636,Z 106,A -132.5032,B 24.9433,C -1.7396,E1 24.9008,E2 218.0944} C_DIS
LIN {X -62.5192,Y -83.0095,Z 106,A -130.2123,B 24.9422,C -1.7567,E1 24.906,E2 215.7544} C_DIS
LIN {X -59.7279,Y -85.0415,Z 106,A -128.8025,B 24.9436,C -1.735,E1 24.9091,E2 214.3915} C_DIS
LIN {X -57.3785,Y -86.6427,Z 106,A -127.197,B 24.9436,C -1.7339,E1 24.9128,E2 212.7832} C_DIS
LIN {X -54.854,Y -88.2627,Z 106,A -125.5029,B 24.9437,C -1.7329,E1 24.9168,E2 211.0862} C_DIS
LIN {X -51.3447,Y -90.3503,Z 106,A -123.0741,B 24.9435,C -1.7363,E1 24.9227,E2 208.6419} C_DIS
LIN {X -47.6576,Y -92.3479,Z 106,A -120.5008,B 24.943,C -1.7433,E1 24.9291,E2 206.045} C_DIS
LIN {X -44.6607,Y -93.8338,Z 106,A -119.3158,B 24.9448,C -1.716,E1 24.932,E2 204.9217} C_DIS
LIN {X -42.2183,Y -94.9584,Z 106,A -117.6949,B 24.9446,C -1.7196,E1 24.9361,E2 203.2885} C_DIS
LIN {X -39.3739,Y -96.1715,Z 106,A -115.8478,B 24.9443,C -1.7232,E1 24.9409,E2 201.4284} C_DIS
LIN {X -36.2634,Y -97.3875,Z 106,A -113.8712,B 24.9441,C -1.7267,E1 24.9461,E2 199.4395} C_DIS
LIN {X -32.9849,Y -98.5457,Z 106,A -112.0412,B 24.9444,C -1.7218,E1 24.9509,E2 197.6177} C_DIS
LIN {X -27.7171,Y -100.1568,Z 106,A -109.1734,B 24.945,C -1.7131,E1 24.9586,E2 194.7657} C_DIS
LIN {X -24.3428,Y -101.0284,Z 106,A -107.1599,B 24.9448,C -1.7156,E1 24.964,E2 192.7434} C_DIS
LIN {X -19.0517,Y -102.1598,Z 106,A -104.1339,B 24.9448,C -1.7159,E1 24.9723,E2 189.713} C_DIS
LIN {X -15.8429,Y -102.7045,Z 106,A -102.4213,B 24.9451,C -1.7123,E1 24.977,E2 188.0077} C_DIS
LIN {X -12.7819,Y -103.1318,Z 106,A -100.5078,B 24.9445,C -1.7201,E1 24.9824,E2 186.0741} C_DIS
LIN {X -9.2001,Y -103.5118,Z 106,A -98.2745,B 24.9439,C -1.7297,E1 24.9887,E2 183.8169} C_DIS
LIN {X -5.9649,Y -103.7482,Z 106,A -96.9556,B 24.9451,C -1.7113,E1 24.9922,E2 182.5413} C_DIS
LIN {X -2.9122,Y -103.8788,Z 106,A -95.2872,B 24.9451,C -1.7108,E1 24.9969,E2 180.8736} C_DIS
LIN {X 0.7371,Y -103.9038,Z 106,A -93.8619,B 24.9466,C -1.6884,E1 25.0007,E2 179.5014} C_DIS
Enddeposition()
LIN {X 0.7371,Y -103.9038,Z 106,A -93.8619,B 24.9466,C -1.6884,E1 25.0007,E2 179.5014} C_DIS
Startdeposition()
$VEL.CP = VEL_PRINT
LIN {X -0.7439,Y -102.944,Z 106,A -94.8926,B 24.946,C -1.6971,E1 24.9979,E2 180.5115} C_DIS
LIN {X -4.8707,Y -102.8324,Z 106,A -97.236,B 24.9462,C -1.6951,E1 24.9913,E2 182.8601} C_DIS
LIN {X -8.3565,Y -102.6071,Z 106,A -99.2183,B 24.9462,C -1.6937,E1 24.9858,E2 184.8466} C_DIS
LIN {X -12.3556,Y -102.2032,Z 106,A -101.2616,B 24.9458,C -1.7013,E1 24.9802,E2 186.873} C_DIS
LIN {X -15.4044,Y -101.7882,Z 106,A -102.9498,B 24.9457,C -1.7026,E1 24.9755,E2 188.5594} C_DIS
LIN {X -18.4586,Y -101.2786,Z 106,A -104.6646,B 24.9457,C -1.7035,E1 24.9708,E2 190.2738} C_DIS
LIN {X -21.1196,Y -100.7579,Z 106,A -106.4254,B 24.9462,C -1.6946,E1 24.9659,E2 192.0578} C_DIS
LIN {X -24.9908,Y -99.8692,Z 106,A -108.6444,B 24.9462,C -1.6954,E1 24.9599,E2 194.2778} C_DIS
LIN {X -31.0071,Y -98.1676,Z 106,A -112.1028,B 24.9459,C -1.6986,E1 24.9506,E2 197.7344} C_DIS
LIN {X -34.7377,Y -96.9102,Z 106,A -114.2541,B 24.9457,C -1.702,E1 24.9449,E2 199.8818} C_DIS
LIN {X -37.1964,Y -95.9931,Z 106,A -115.5001,B 24.9451,C -1.7113,E1 24.9417,E2 201.1083} C_DIS
LIN {X -40.3814,Y -94.6972,Z 106,A -117.5756,B 24.9454,C -1.7073,E1 24.9364,E2 203.1981} C_DIS
LIN {X -43.5242,Y -93.2935,Z 106,A -119.5226,B 24.9454,C -1.7083,E1 24.9314,E2 205.1475} C_DIS
LIN {X -46.756,Y -91.7164,Z 106,A -121.5127,B 24.9451,C -1.7112,E1 24.9264,E2 207.136} C_DIS
LIN {X -48.9217,Y -90.5799,Z 106,A -123.2691,B 24.9459,C -1.6985,E1 24.922,E2 208.9273} C_DIS
LIN {X -51.7193,Y -89.0134,Z 106,A -124.8688,B 24.9453,C -1.7078,E1 24.9182,E2 210.5098} C_DIS
LIN {X -55.4123,Y -86.7615,Z 106,A -126.7896,B 24.944,C -1.7292,E1 24.9137,E2 212.3857} C_DIS
LIN {X -57.0886,Y -85.6689,Z 106,A -128.3304,B 24.9449,C -1.7154,E1 24.9101,E2 213.9645} C_DIS
LIN {X -60.2276,Y -83.4922,Z 106,A -130.4275,B 24.9446,C -1.72,E1 24.9053,E2 216.0578} C_DIS
Enddeposition()
END
